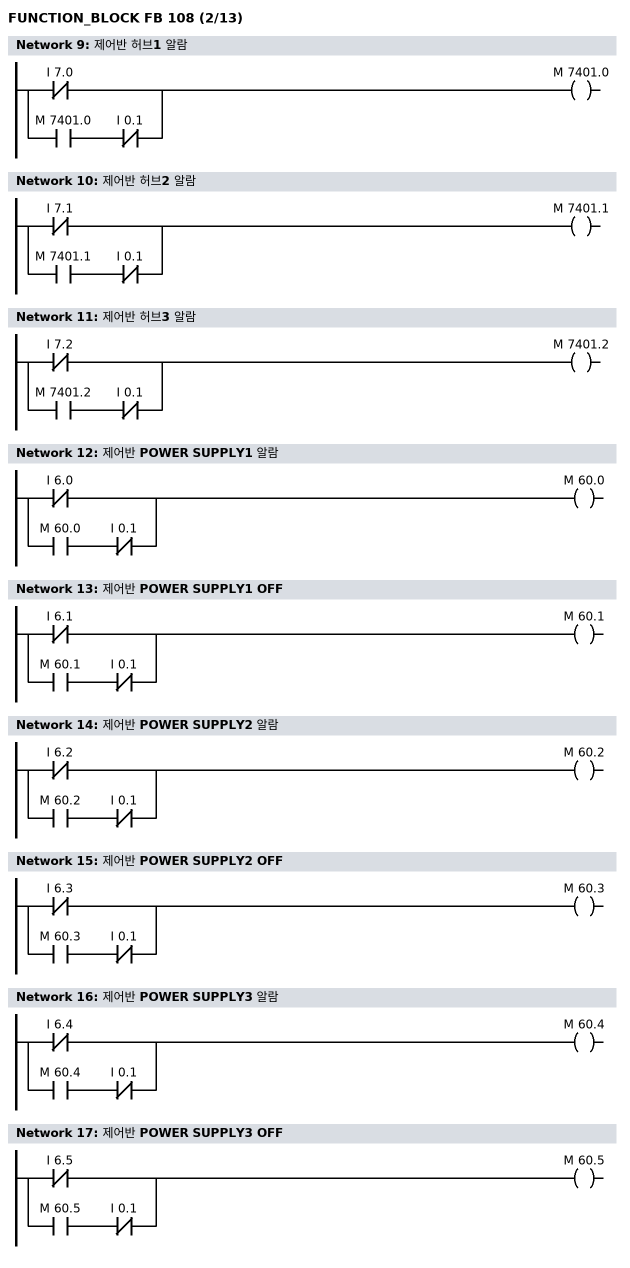

      ON    I      7.0;
      O     ;
      A     M   7401.0;
      AN    I      0.1;
      =     M   7401.0;
NETWORK
TITLE =제어반 허브2 알람

      ON    I      7.1;
      O     ;
      A     M   7401.1;
      AN    I      0.1;
      =     M   7401.1;
NETWORK
TITLE =제어반 허브3 알람

      ON    I      7.2;
      O     ;
      A     M   7401.2;
      AN    I      0.1;
      =     M   7401.2;
NETWORK
TITLE =제어반 POWER SUPPLY1 알람

      ON    I      6.0;
      O     ;
      A     M     60.0;
      AN    I      0.1;
      =     M     60.0;
NETWORK
TITLE =제어반 POWER SUPPLY1 OFF

      ON    I      6.1;
      O     ;
      A     M     60.1;
      AN    I      0.1;
      =     M     60.1;
NETWORK
TITLE =제어반 POWER SUPPLY2 알람
//
//
      ON    I      6.2;
      O     ;
      A     M     60.2;
      AN    I      0.1;
      =     M     60.2;
NETWORK
TITLE =제어반 POWER SUPPLY2 OFF

      ON    I      6.3;
      O     ;
      A     M     60.3;
      AN    I      0.1;
      =     M     60.3;
NETWORK
TITLE =제어반 POWER SUPPLY3 알람
//
//
      ON    I      6.4;
      O     ;
      A     M     60.4;
      AN    I      0.1;
      =     M     60.4;
NETWORK
TITLE =제어반 POWER SUPPLY3 OFF

      ON    I      6.5;
      O     ;
      A     M     60.5;
      AN    I      0.1;
      =     M     60.5;
NETWORK
TITLE =제어반 서지보호기 알람
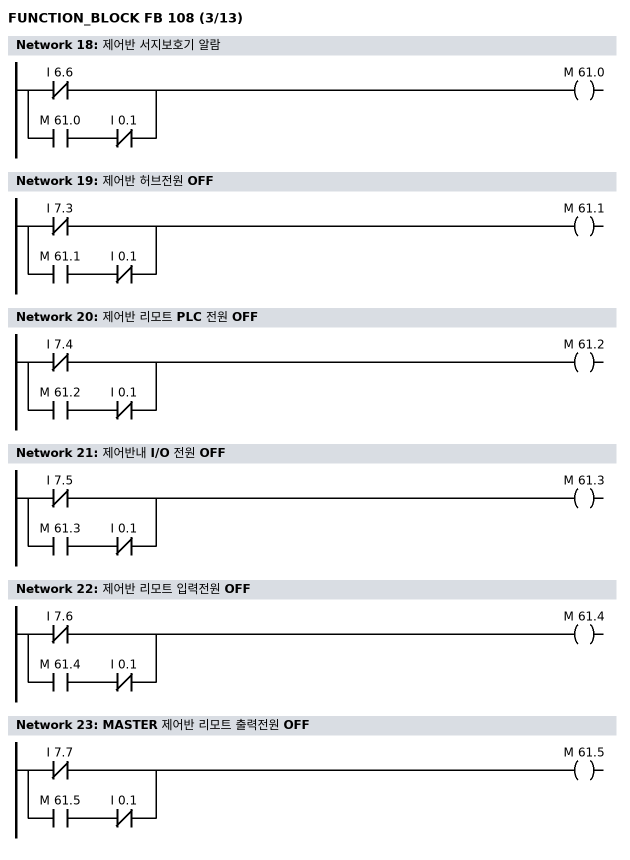

      ON    I      6.6;
      O     ;
      A     M     61.0;
      AN    I      0.1;
      =     M     61.0;
NETWORK
TITLE =제어반 허브전원 OFF

      ON    I      7.3;
      O     ;
      A     M     61.1;
      AN    I      0.1;
      =     M     61.1;
NETWORK
TITLE =제어반 리모트 PLC 전원 OFF

      ON    I      7.4;
      O     ;
      A     M     61.2;
      AN    I      0.1;
      =     M     61.2;
NETWORK
TITLE =제어반내 I/O 전원 OFF

      ON    I      7.5;
      O     ;
      A     M     61.3;
      AN    I      0.1;
      =     M     61.3;
NETWORK
TITLE =제어반 리모트 입력전원 OFF

      ON    I      7.6;
      O     ;
      A     M     61.4;
      AN    I      0.1;
      =     M     61.4;
NETWORK
TITLE =MASTER 제어반 리모트 출력전원 OFF

      ON    I      7.7;
      O     ;
      A     M     61.5;
      AN    I      0.1;
      =     M     61.5;
NETWORK
TITLE =PROFINET ALARM-모듈이상이나 통신케이블단선(1~10)
//
//
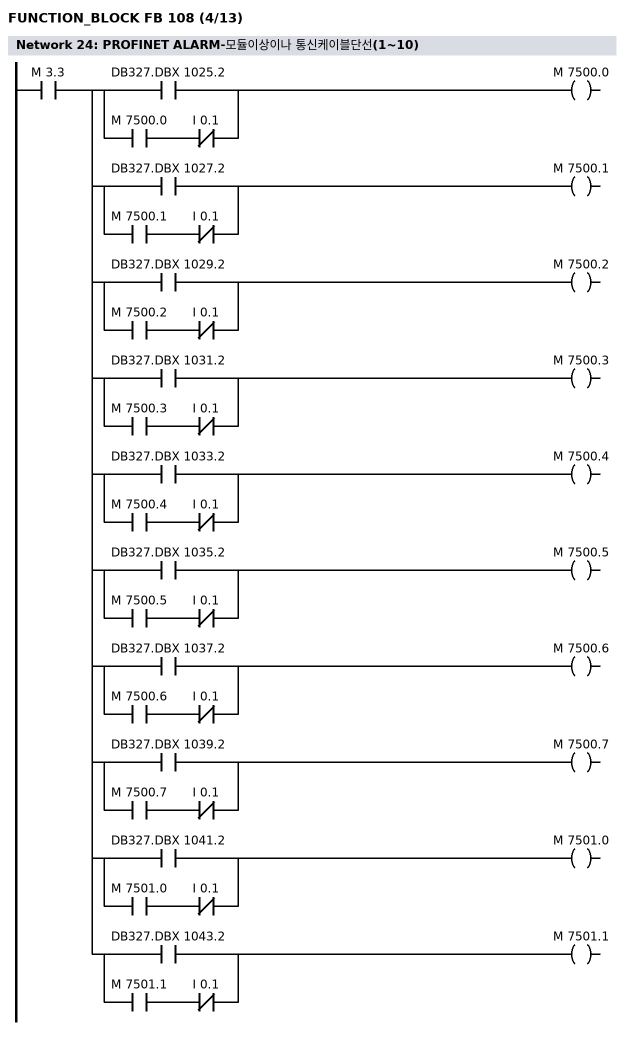
      A     M      3.3;
      =     L      0.0;
      A     L      0.0;
      A(    ;
      O     DB327.DBX 1025.2;
      O     ;
      A     M   7500.0;
      AN    I      0.1;
      )     ;
      =     M   7500.0;
      A     L      0.0;
      A(    ;
      O     DB327.DBX 1027.2;
      O     ;
      A     M   7500.1;
      AN    I      0.1;
      )     ;
      =     M   7500.1;
      A     L      0.0;
      A(    ;
      O     DB327.DBX 1029.2;
      O     ;
      A     M   7500.2;
      AN    I      0.1;
      )     ;
      =     M   7500.2;
      A     L      0.0;
      A(    ;
      O     DB327.DBX 1031.2;
      O     ;
      A     M   7500.3;
      AN    I      0.1;
      )     ;
      =     M   7500.3;
      A     L      0.0;
      A(    ;
      O     DB327.DBX 1033.2;
      O     ;
      A     M   7500.4;
      AN    I      0.1;
      )     ;
      =     M   7500.4;
      A     L      0.0;
      A(    ;
      O     DB327.DBX 1035.2;
      O     ;
      A     M   7500.5;
      AN    I      0.1;
      )     ;
      =     M   7500.5;
      A     L      0.0;
      A(    ;
      O     DB327.DBX 1037.2;
      O     ;
      A     M   7500.6;
      AN    I      0.1;
      )     ;
      =     M   7500.6;
      A     L      0.0;
      A(    ;
      O     DB327.DBX 1039.2;
      O     ;
      A     M   7500.7;
      AN    I      0.1;
      )     ;
      =     M   7500.7;
      A     L      0.0;
      A(    ;
      O     DB327.DBX 1041.2;
      O     ;
      A     M   7501.0;
      AN    I      0.1;
      )     ;
      =     M   7501.0;
      A     L      0.0;
      A(    ;
      O     DB327.DBX 1043.2;
      O     ;
      A     M   7501.1;
      AN    I      0.1;
      )     ;
      =     M   7501.1;
NETWORK
TITLE =PROFINET ALARM-모듈이상이나 통신케이블단선(11~20)
//
//
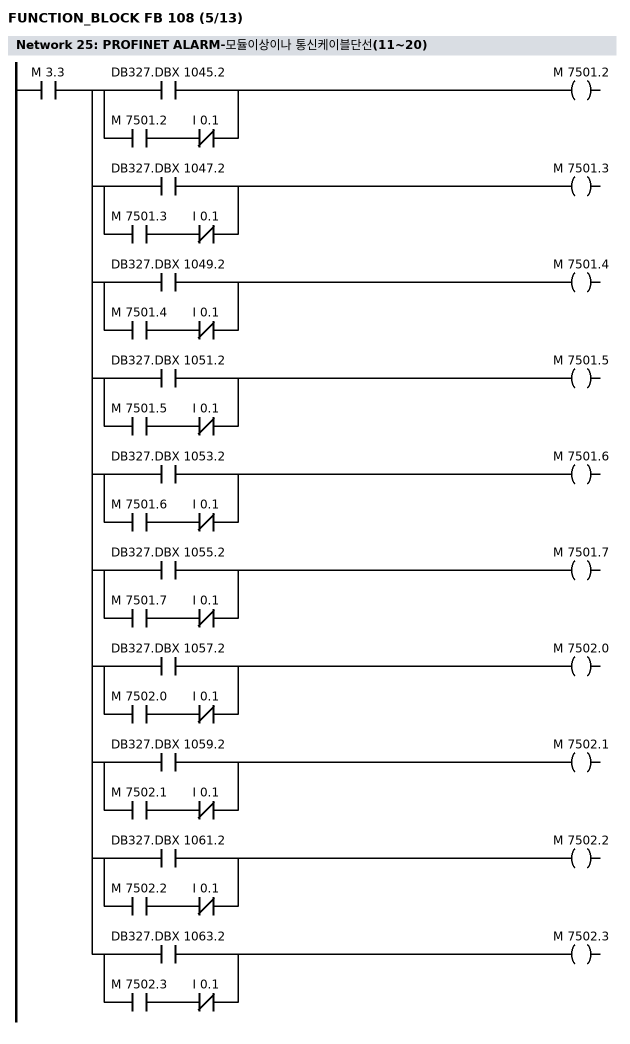
      A     M      3.3;
      =     L      0.0;
      A     L      0.0;
      A(    ;
      O     DB327.DBX 1045.2;
      O     ;
      A     M   7501.2;
      AN    I      0.1;
      )     ;
      =     M   7501.2;
      A     L      0.0;
      A(    ;
      O     DB327.DBX 1047.2;
      O     ;
      A     M   7501.3;
      AN    I      0.1;
      )     ;
      =     M   7501.3;
      A     L      0.0;
      A(    ;
      O     DB327.DBX 1049.2;
      O     ;
      A     M   7501.4;
      AN    I      0.1;
      )     ;
      =     M   7501.4;
      A     L      0.0;
      A(    ;
      O     DB327.DBX 1051.2;
      O     ;
      A     M   7501.5;
      AN    I      0.1;
      )     ;
      =     M   7501.5;
      A     L      0.0;
      A(    ;
      O     DB327.DBX 1053.2;
      O     ;
      A     M   7501.6;
      AN    I      0.1;
      )     ;
      =     M   7501.6;
      A     L      0.0;
      A(    ;
      O     DB327.DBX 1055.2;
      O     ;
      A     M   7501.7;
      AN    I      0.1;
      )     ;
      =     M   7501.7;
      A     L      0.0;
      A(    ;
      O     DB327.DBX 1057.2;
      O     ;
      A     M   7502.0;
      AN    I      0.1;
      )     ;
      =     M   7502.0;
      A     L      0.0;
      A(    ;
      O     DB327.DBX 1059.2;
      O     ;
      A     M   7502.1;
      AN    I      0.1;
      )     ;
      =     M   7502.1;
      A     L      0.0;
      A(    ;
      O     DB327.DBX 1061.2;
      O     ;
      A     M   7502.2;
      AN    I      0.1;
      )     ;
      =     M   7502.2;
      A     L      0.0;
      A(    ;
      O     DB327.DBX 1063.2;
      O     ;
      A     M   7502.3;
      AN    I      0.1;
      )     ;
      =     M   7502.3;
NETWORK
TITLE =PROFINET ALARM-모듈이상이나 통신케이블단선(21~30)
//
//
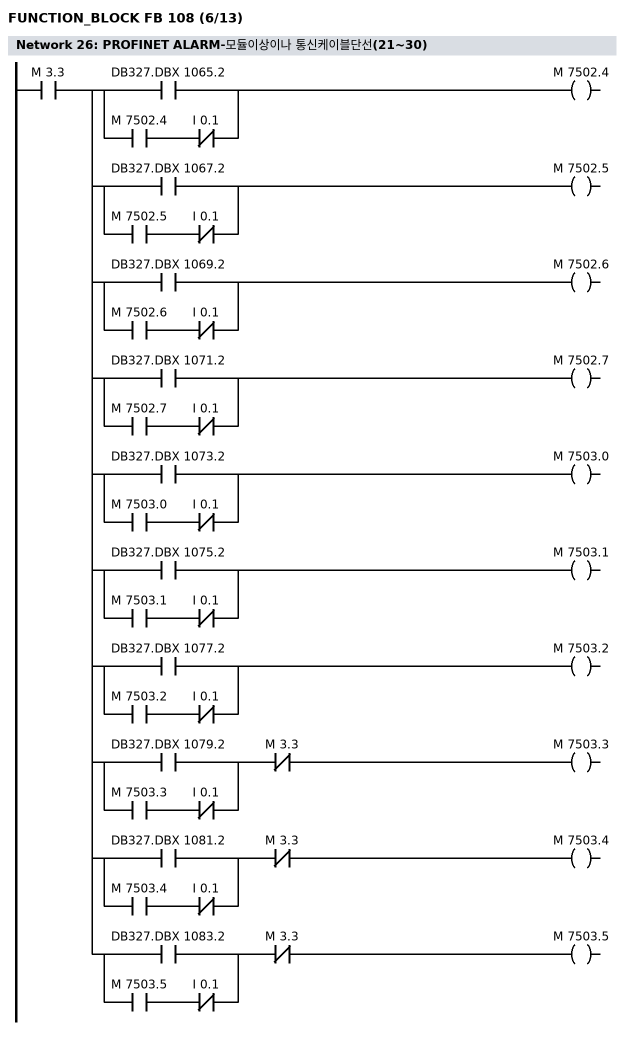
      A     M      3.3;
      =     L      0.0;
      A     L      0.0;
      A(    ;
      O     DB327.DBX 1065.2;
      O     ;
      A     M   7502.4;
      AN    I      0.1;
      )     ;
      =     M   7502.4;
      A     L      0.0;
      A(    ;
      O     DB327.DBX 1067.2;
      O     ;
      A     M   7502.5;
      AN    I      0.1;
      )     ;
      =     M   7502.5;
      A     L      0.0;
      A(    ;
      O     DB327.DBX 1069.2;
      O     ;
      A     M   7502.6;
      AN    I      0.1;
      )     ;
      =     M   7502.6;
      A     L      0.0;
      A(    ;
      O     DB327.DBX 1071.2;
      O     ;
      A     M   7502.7;
      AN    I      0.1;
      )     ;
      =     M   7502.7;
      A     L      0.0;
      A(    ;
      O     DB327.DBX 1073.2;
      O     ;
      A     M   7503.0;
      AN    I      0.1;
      )     ;
      =     M   7503.0;
      A     L      0.0;
      A(    ;
      O     DB327.DBX 1075.2;
      O     ;
      A     M   7503.1;
      AN    I      0.1;
      )     ;
      =     M   7503.1;
      A     L      0.0;
      A(    ;
      O     DB327.DBX 1077.2;
      O     ;
      A     M   7503.2;
      AN    I      0.1;
      )     ;
      =     M   7503.2;
      A     L      0.0;
      A(    ;
      O     DB327.DBX 1079.2;
      O     ;
      A     M   7503.3;
      AN    I      0.1;
      )     ;
      AN    M      3.3;
      =     M   7503.3;
      A     L      0.0;
      A(    ;
      O     DB327.DBX 1081.2;
      O     ;
      A     M   7503.4;
      AN    I      0.1;
      )     ;
      AN    M      3.3;
      =     M   7503.4;
      A     L      0.0;
      A(    ;
      O     DB327.DBX 1083.2;
      O     ;
      A     M   7503.5;
      AN    I      0.1;
      )     ;
      AN    M      3.3;
      =     M   7503.5;
NETWORK
TITLE =PROFINET ALARM-모듈이상이나 통신케이블단선(31~40)
//
//
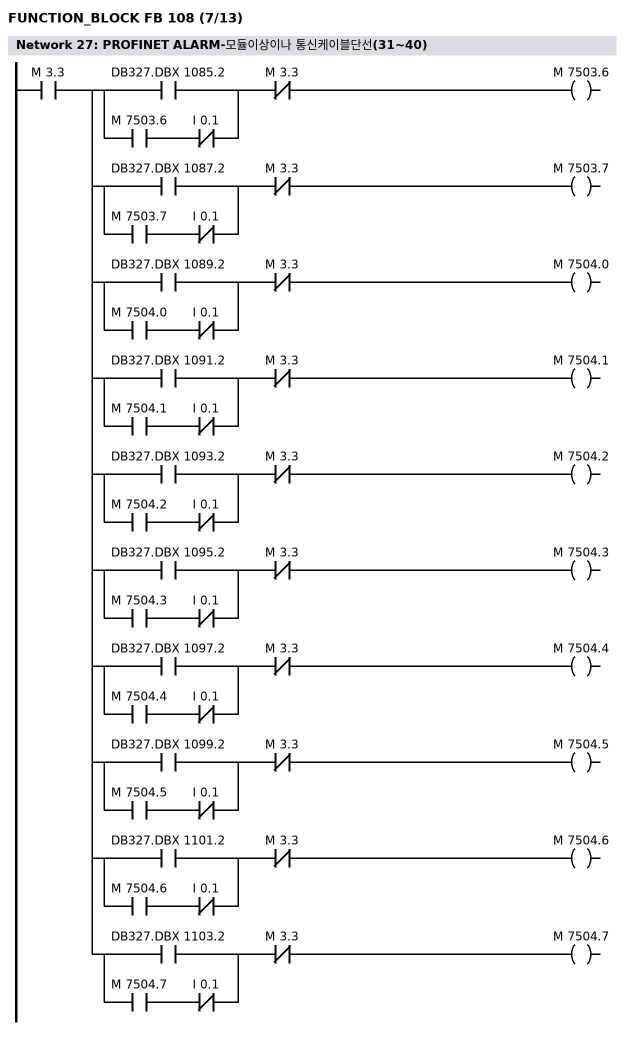
      A     M      3.3;
      =     L      0.0;
      A     L      0.0;
      A(    ;
      O     DB327.DBX 1085.2;
      O     ;
      A     M   7503.6;
      AN    I      0.1;
      )     ;
      AN    M      3.3;
      =     M   7503.6;
      A     L      0.0;
      A(    ;
      O     DB327.DBX 1087.2;
      O     ;
      A     M   7503.7;
      AN    I      0.1;
      )     ;
      AN    M      3.3;
      =     M   7503.7;
      A     L      0.0;
      A(    ;
      O     DB327.DBX 1089.2;
      O     ;
      A     M   7504.0;
      AN    I      0.1;
      )     ;
      AN    M      3.3;
      =     M   7504.0;
      A     L      0.0;
      A(    ;
      O     DB327.DBX 1091.2;
      O     ;
      A     M   7504.1;
      AN    I      0.1;
      )     ;
      AN    M      3.3;
      =     M   7504.1;
      A     L      0.0;
      A(    ;
      O     DB327.DBX 1093.2;
      O     ;
      A     M   7504.2;
      AN    I      0.1;
      )     ;
      AN    M      3.3;
      =     M   7504.2;
      A     L      0.0;
      A(    ;
      O     DB327.DBX 1095.2;
      O     ;
      A     M   7504.3;
      AN    I      0.1;
      )     ;
      AN    M      3.3;
      =     M   7504.3;
      A     L      0.0;
      A(    ;
      O     DB327.DBX 1097.2;
      O     ;
      A     M   7504.4;
      AN    I      0.1;
      )     ;
      AN    M      3.3;
      =     M   7504.4;
      A     L      0.0;
      A(    ;
      O     DB327.DBX 1099.2;
      O     ;
      A     M   7504.5;
      AN    I      0.1;
      )     ;
      AN    M      3.3;
      =     M   7504.5;
      A     L      0.0;
      A(    ;
      O     DB327.DBX 1101.2;
      O     ;
      A     M   7504.6;
      AN    I      0.1;
      )     ;
      AN    M      3.3;
      =     M   7504.6;
      A     L      0.0;
      A(    ;
      O     DB327.DBX 1103.2;
      O     ;
      A     M   7504.7;
      AN    I      0.1;
      )     ;
      AN    M      3.3;
      =     M   7504.7;
NETWORK
TITLE =PROFINET ALARM-모듈이상이나 통신케이블단선(150~159)
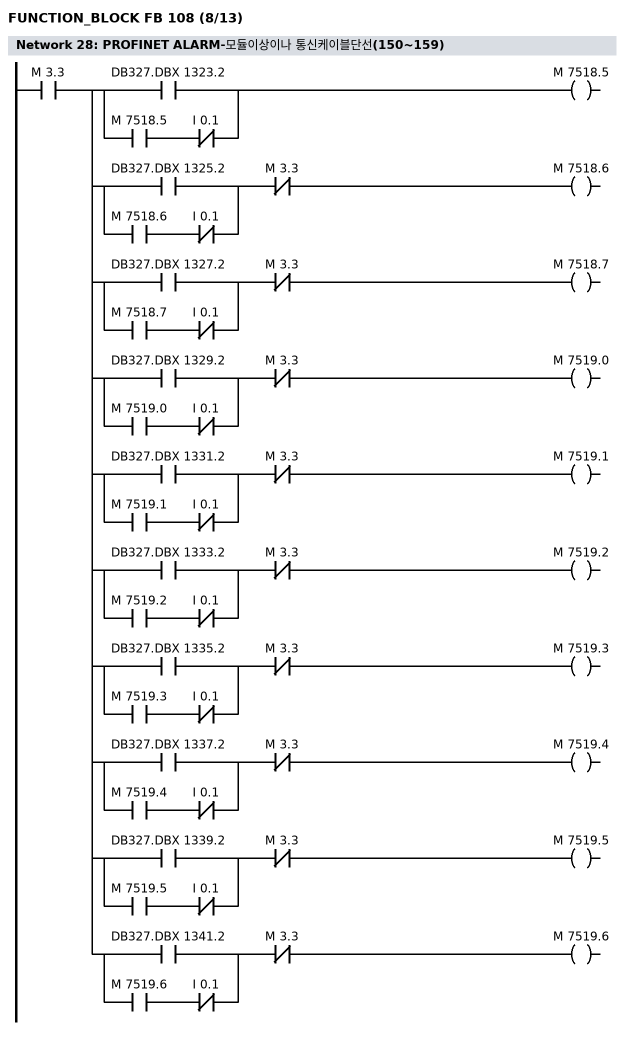

      A     M      3.3;
      =     L      0.0;
      A     L      0.0;
      A(    ;
      O     DB327.DBX 1323.2;
      O     ;
      A     M   7518.5;
      AN    I      0.1;
      )     ;
      =     M   7518.5;
      A     L      0.0;
      A(    ;
      O     DB327.DBX 1325.2;
      O     ;
      A     M   7518.6;
      AN    I      0.1;
      )     ;
      AN    M      3.3;
      =     M   7518.6;
      A     L      0.0;
      A(    ;
      O     DB327.DBX 1327.2;
      O     ;
      A     M   7518.7;
      AN    I      0.1;
      )     ;
      AN    M      3.3;
      =     M   7518.7;
      A     L      0.0;
      A(    ;
      O     DB327.DBX 1329.2;
      O     ;
      A     M   7519.0;
      AN    I      0.1;
      )     ;
      AN    M      3.3;
      =     M   7519.0;
      A     L      0.0;
      A(    ;
      O     DB327.DBX 1331.2;
      O     ;
      A     M   7519.1;
      AN    I      0.1;
      )     ;
      AN    M      3.3;
      =     M   7519.1;
      A     L      0.0;
      A(    ;
      O     DB327.DBX 1333.2;
      O     ;
      A     M   7519.2;
      AN    I      0.1;
      )     ;
      AN    M      3.3;
      =     M   7519.2;
      A     L      0.0;
      A(    ;
      O     DB327.DBX 1335.2;
      O     ;
      A     M   7519.3;
      AN    I      0.1;
      )     ;
      AN    M      3.3;
      =     M   7519.3;
      A     L      0.0;
      A(    ;
      O     DB327.DBX 1337.2;
      O     ;
      A     M   7519.4;
      AN    I      0.1;
      )     ;
      AN    M      3.3;
      =     M   7519.4;
      A     L      0.0;
      A(    ;
      O     DB327.DBX 1339.2;
      O     ;
      A     M   7519.5;
      AN    I      0.1;
      )     ;
      AN    M      3.3;
      =     M   7519.5;
      A     L      0.0;
      A(    ;
      O     DB327.DBX 1341.2;
      O     ;
      A     M   7519.6;
      AN    I      0.1;
      )     ;
      AN    M      3.3;
      =     M   7519.6;
NETWORK
TITLE =PROFINET MODULE ERROR(1~10)
//
//
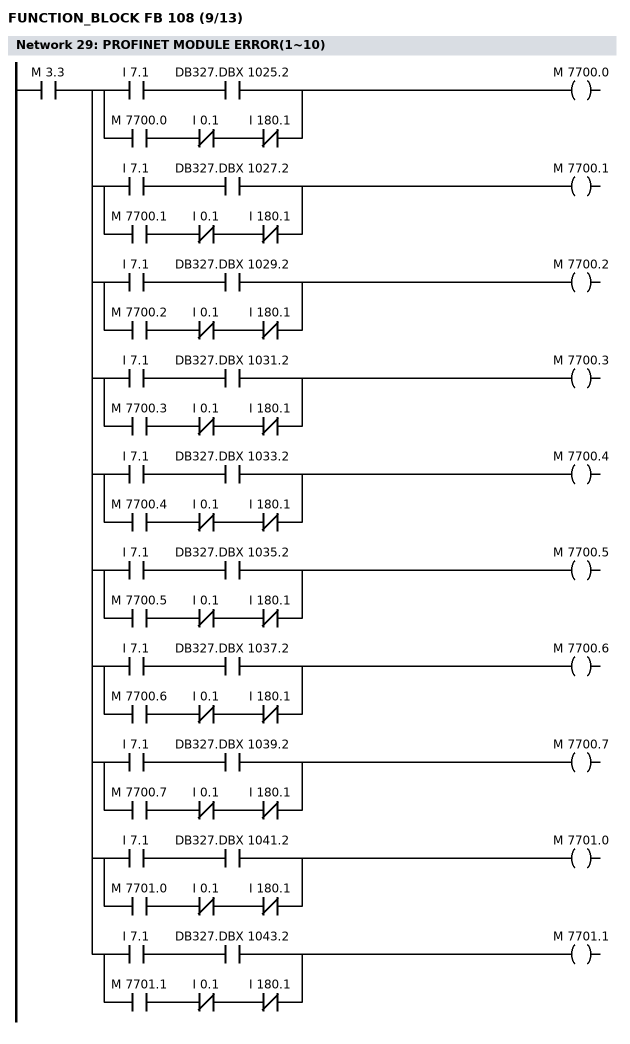
      A     M      3.3;
      =     L      0.0;
      A     L      0.0;
      A(    ;
      A     I      7.1;
      A     DB327.DBX 1025.2;
      O     ;
      A     M   7700.0;
      AN    I      0.1;
      AN    I    180.1;
      )     ;
      =     M   7700.0;
      A     L      0.0;
      A(    ;
      A     I      7.1;
      A     DB327.DBX 1027.2;
      O     ;
      A     M   7700.1;
      AN    I      0.1;
      AN    I    180.1;
      )     ;
      =     M   7700.1;
      A     L      0.0;
      A(    ;
      A     I      7.1;
      A     DB327.DBX 1029.2;
      O     ;
      A     M   7700.2;
      AN    I      0.1;
      AN    I    180.1;
      )     ;
      =     M   7700.2;
      A     L      0.0;
      A(    ;
      A     I      7.1;
      A     DB327.DBX 1031.2;
      O     ;
      A     M   7700.3;
      AN    I      0.1;
      AN    I    180.1;
      )     ;
      =     M   7700.3;
      A     L      0.0;
      A(    ;
      A     I      7.1;
      A     DB327.DBX 1033.2;
      O     ;
      A     M   7700.4;
      AN    I      0.1;
      AN    I    180.1;
      )     ;
      =     M   7700.4;
      A     L      0.0;
      A(    ;
      A     I      7.1;
      A     DB327.DBX 1035.2;
      O     ;
      A     M   7700.5;
      AN    I      0.1;
      AN    I    180.1;
      )     ;
      =     M   7700.5;
      A     L      0.0;
      A(    ;
      A     I      7.1;
      A     DB327.DBX 1037.2;
      O     ;
      A     M   7700.6;
      AN    I      0.1;
      AN    I    180.1;
      )     ;
      =     M   7700.6;
      A     L      0.0;
      A(    ;
      A     I      7.1;
      A     DB327.DBX 1039.2;
      O     ;
      A     M   7700.7;
      AN    I      0.1;
      AN    I    180.1;
      )     ;
      =     M   7700.7;
      A     L      0.0;
      A(    ;
      A     I      7.1;
      A     DB327.DBX 1041.2;
      O     ;
      A     M   7701.0;
      AN    I      0.1;
      AN    I    180.1;
      )     ;
      =     M   7701.0;
      A     L      0.0;
      A(    ;
      A     I      7.1;
      A     DB327.DBX 1043.2;
      O     ;
      A     M   7701.1;
      AN    I      0.1;
      AN    I    180.1;
      )     ;
      =     M   7701.1;
NETWORK
TITLE =PROFINET MODULE ERROR(11~20)
//
//
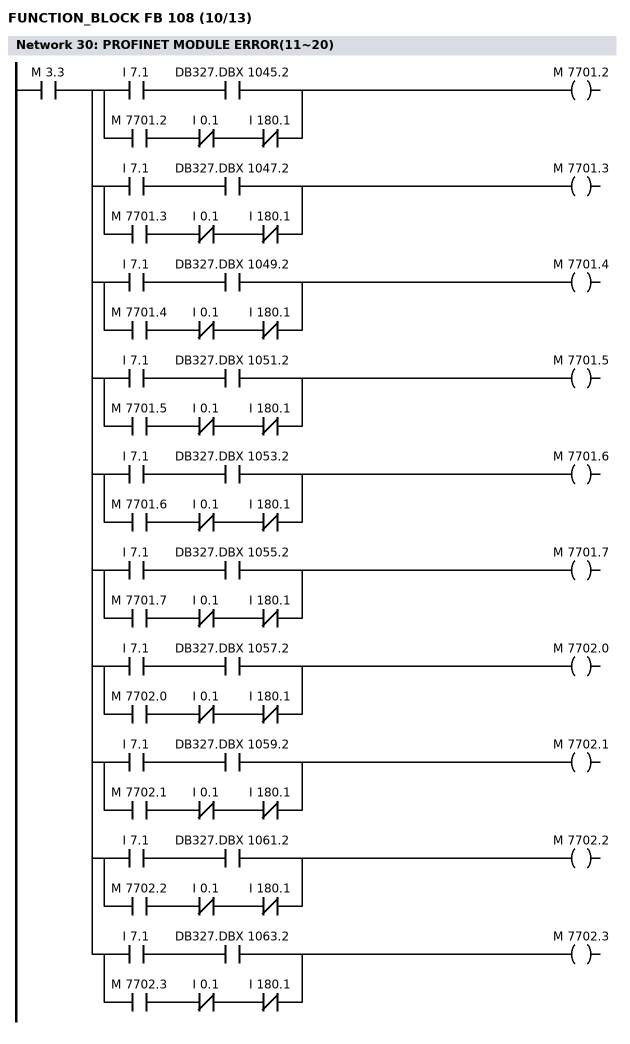
      A     M      3.3;
      =     L      0.0;
      A     L      0.0;
      A(    ;
      A     I      7.1;
      A     DB327.DBX 1045.2;
      O     ;
      A     M   7701.2;
      AN    I      0.1;
      AN    I    180.1;
      )     ;
      =     M   7701.2;
      A     L      0.0;
      A(    ;
      A     I      7.1;
      A     DB327.DBX 1047.2;
      O     ;
      A     M   7701.3;
      AN    I      0.1;
      AN    I    180.1;
      )     ;
      =     M   7701.3;
      A     L      0.0;
      A(    ;
      A     I      7.1;
      A     DB327.DBX 1049.2;
      O     ;
      A     M   7701.4;
      AN    I      0.1;
      AN    I    180.1;
      )     ;
      =     M   7701.4;
      A     L      0.0;
      A(    ;
      A     I      7.1;
      A     DB327.DBX 1051.2;
      O     ;
      A     M   7701.5;
      AN    I      0.1;
      AN    I    180.1;
      )     ;
      =     M   7701.5;
      A     L      0.0;
      A(    ;
      A     I      7.1;
      A     DB327.DBX 1053.2;
      O     ;
      A     M   7701.6;
      AN    I      0.1;
      AN    I    180.1;
      )     ;
      =     M   7701.6;
      A     L      0.0;
      A(    ;
      A     I      7.1;
      A     DB327.DBX 1055.2;
      O     ;
      A     M   7701.7;
      AN    I      0.1;
      AN    I    180.1;
      )     ;
      =     M   7701.7;
      A     L      0.0;
      A(    ;
      A     I      7.1;
      A     DB327.DBX 1057.2;
      O     ;
      A     M   7702.0;
      AN    I      0.1;
      AN    I    180.1;
      )     ;
      =     M   7702.0;
      A     L      0.0;
      A(    ;
      A     I      7.1;
      A     DB327.DBX 1059.2;
      O     ;
      A     M   7702.1;
      AN    I      0.1;
      AN    I    180.1;
      )     ;
      =     M   7702.1;
      A     L      0.0;
      A(    ;
      A     I      7.1;
      A     DB327.DBX 1061.2;
      O     ;
      A     M   7702.2;
      AN    I      0.1;
      AN    I    180.1;
      )     ;
      =     M   7702.2;
      A     L      0.0;
      A(    ;
      A     I      7.1;
      A     DB327.DBX 1063.2;
      O     ;
      A     M   7702.3;
      AN    I      0.1;
      AN    I    180.1;
      )     ;
      =     M   7702.3;
NETWORK
TITLE =PROFINET MODULE ERROR(21~30)
//
//
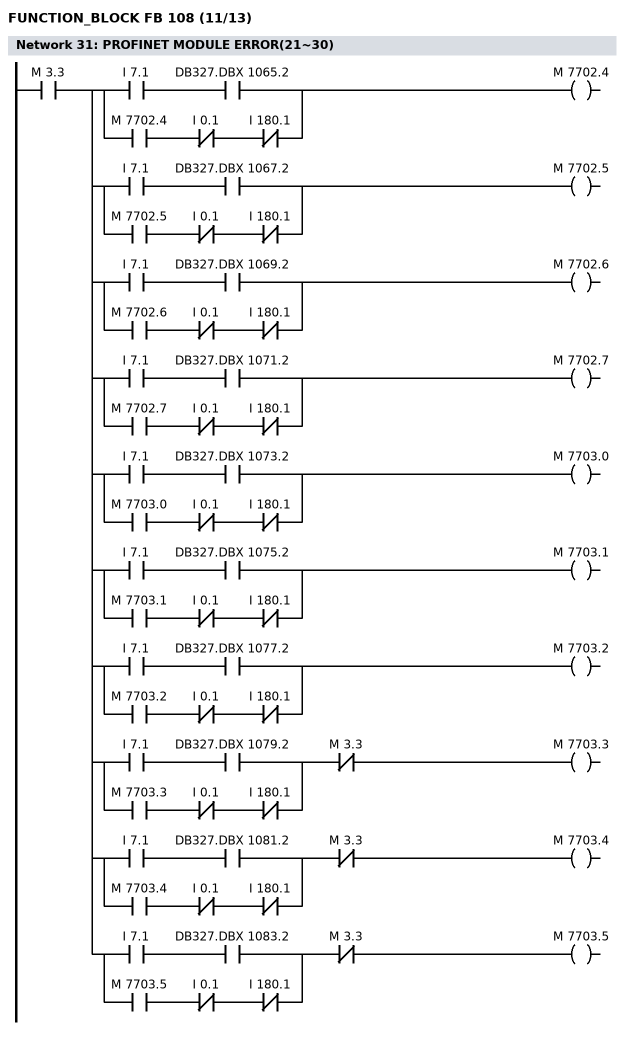
      A     M      3.3;
      =     L      0.0;
      A     L      0.0;
      A(    ;
      A     I      7.1;
      A     DB327.DBX 1065.2;
      O     ;
      A     M   7702.4;
      AN    I      0.1;
      AN    I    180.1;
      )     ;
      =     M   7702.4;
      A     L      0.0;
      A(    ;
      A     I      7.1;
      A     DB327.DBX 1067.2;
      O     ;
      A     M   7702.5;
      AN    I      0.1;
      AN    I    180.1;
      )     ;
      =     M   7702.5;
      A     L      0.0;
      A(    ;
      A     I      7.1;
      A     DB327.DBX 1069.2;
      O     ;
      A     M   7702.6;
      AN    I      0.1;
      AN    I    180.1;
      )     ;
      =     M   7702.6;
      A     L      0.0;
      A(    ;
      A     I      7.1;
      A     DB327.DBX 1071.2;
      O     ;
      A     M   7702.7;
      AN    I      0.1;
      AN    I    180.1;
      )     ;
      =     M   7702.7;
      A     L      0.0;
      A(    ;
      A     I      7.1;
      A     DB327.DBX 1073.2;
      O     ;
      A     M   7703.0;
      AN    I      0.1;
      AN    I    180.1;
      )     ;
      =     M   7703.0;
      A     L      0.0;
      A(    ;
      A     I      7.1;
      A     DB327.DBX 1075.2;
      O     ;
      A     M   7703.1;
      AN    I      0.1;
      AN    I    180.1;
      )     ;
      =     M   7703.1;
      A     L      0.0;
      A(    ;
      A     I      7.1;
      A     DB327.DBX 1077.2;
      O     ;
      A     M   7703.2;
      AN    I      0.1;
      AN    I    180.1;
      )     ;
      =     M   7703.2;
      A     L      0.0;
      A(    ;
      A     I      7.1;
      A     DB327.DBX 1079.2;
      O     ;
      A     M   7703.3;
      AN    I      0.1;
      AN    I    180.1;
      )     ;
      AN    M      3.3;
      =     M   7703.3;
      A     L      0.0;
      A(    ;
      A     I      7.1;
      A     DB327.DBX 1081.2;
      O     ;
      A     M   7703.4;
      AN    I      0.1;
      AN    I    180.1;
      )     ;
      AN    M      3.3;
      =     M   7703.4;
      A     L      0.0;
      A(    ;
      A     I      7.1;
      A     DB327.DBX 1083.2;
      O     ;
      A     M   7703.5;
      AN    I      0.1;
      AN    I    180.1;
      )     ;
      AN    M      3.3;
      =     M   7703.5;
NETWORK
TITLE =PROFINET MODULE ERROR(31~40)
//
//
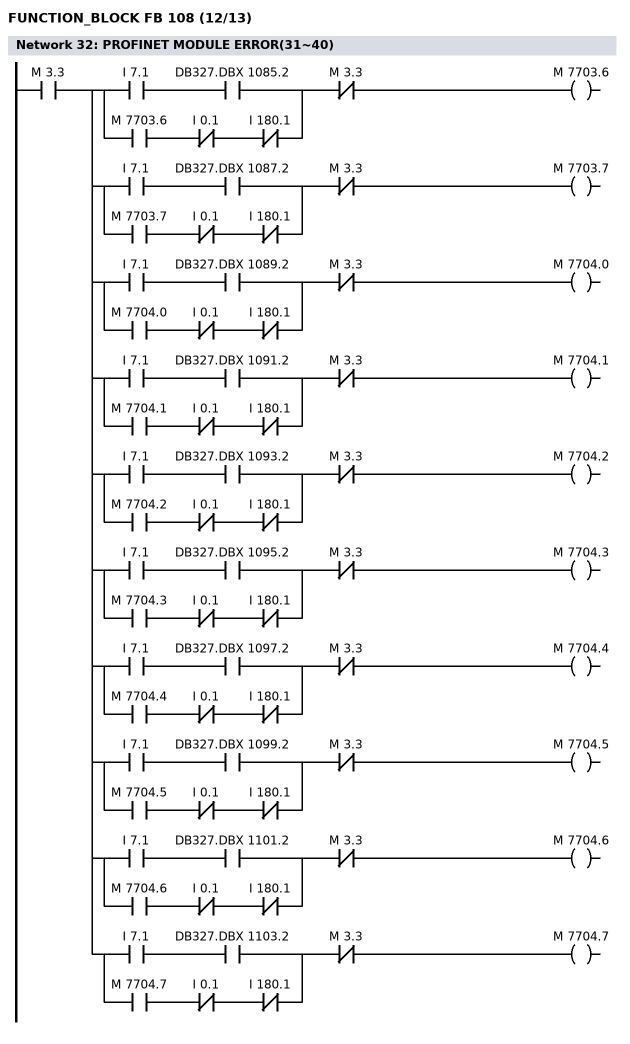
      A     M      3.3;
      =     L      0.0;
      A     L      0.0;
      A(    ;
      A     I      7.1;
      A     DB327.DBX 1085.2;
      O     ;
      A     M   7703.6;
      AN    I      0.1;
      AN    I    180.1;
      )     ;
      AN    M      3.3;
      =     M   7703.6;
      A     L      0.0;
      A(    ;
      A     I      7.1;
      A     DB327.DBX 1087.2;
      O     ;
      A     M   7703.7;
      AN    I      0.1;
      AN    I    180.1;
      )     ;
      AN    M      3.3;
      =     M   7703.7;
      A     L      0.0;
      A(    ;
      A     I      7.1;
      A     DB327.DBX 1089.2;
      O     ;
      A     M   7704.0;
      AN    I      0.1;
      AN    I    180.1;
      )     ;
      AN    M      3.3;
      =     M   7704.0;
      A     L      0.0;
      A(    ;
      A     I      7.1;
      A     DB327.DBX 1091.2;
      O     ;
      A     M   7704.1;
      AN    I      0.1;
      AN    I    180.1;
      )     ;
      AN    M      3.3;
      =     M   7704.1;
      A     L      0.0;
      A(    ;
      A     I      7.1;
      A     DB327.DBX 1093.2;
      O     ;
      A     M   7704.2;
      AN    I      0.1;
      AN    I    180.1;
      )     ;
      AN    M      3.3;
      =     M   7704.2;
      A     L      0.0;
      A(    ;
      A     I      7.1;
      A     DB327.DBX 1095.2;
      O     ;
      A     M   7704.3;
      AN    I      0.1;
      AN    I    180.1;
      )     ;
      AN    M      3.3;
      =     M   7704.3;
      A     L      0.0;
      A(    ;
      A     I      7.1;
      A     DB327.DBX 1097.2;
      O     ;
      A     M   7704.4;
      AN    I      0.1;
      AN    I    180.1;
      )     ;
      AN    M      3.3;
      =     M   7704.4;
      A     L      0.0;
      A(    ;
      A     I      7.1;
      A     DB327.DBX 1099.2;
      O     ;
      A     M   7704.5;
      AN    I      0.1;
      AN    I    180.1;
      )     ;
      AN    M      3.3;
      =     M   7704.5;
      A     L      0.0;
      A(    ;
      A     I      7.1;
      A     DB327.DBX 1101.2;
      O     ;
      A     M   7704.6;
      AN    I      0.1;
      AN    I    180.1;
      )     ;
      AN    M      3.3;
      =     M   7704.6;
      A     L      0.0;
      A(    ;
      A     I      7.1;
      A     DB327.DBX 1103.2;
      O     ;
      A     M   7704.7;
      AN    I      0.1;
      AN    I    180.1;
      )     ;
      AN    M      3.3;
      =     M   7704.7;
NETWORK
TITLE =PROFINET MODULE ERROR(150~159)
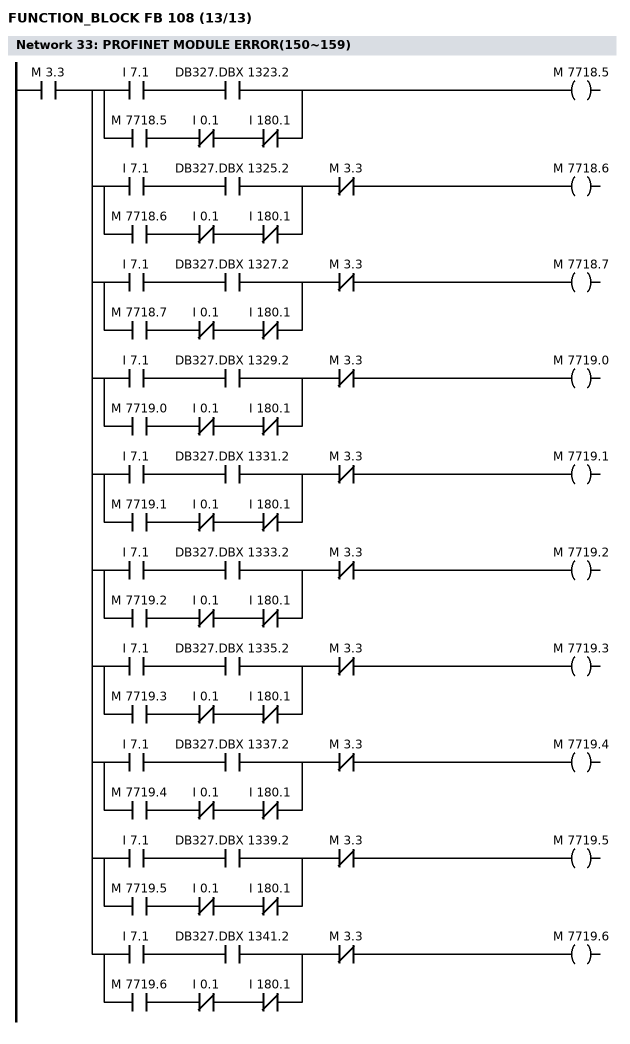

      A     M      3.3;
      =     L      0.0;
      A     L      0.0;
      A(    ;
      A     I      7.1;
      A     DB327.DBX 1323.2;
      O     ;
      A     M   7718.5;
      AN    I      0.1;
      AN    I    180.1;
      )     ;
      =     M   7718.5;
      A     L      0.0;
      A(    ;
      A     I      7.1;
      A     DB327.DBX 1325.2;
      O     ;
      A     M   7718.6;
      AN    I      0.1;
      AN    I    180.1;
      )     ;
      AN    M      3.3;
      =     M   7718.6;
      A     L      0.0;
      A(    ;
      A     I      7.1;
      A     DB327.DBX 1327.2;
      O     ;
      A     M   7718.7;
      AN    I      0.1;
      AN    I    180.1;
      )     ;
      AN    M      3.3;
      =     M   7718.7;
      A     L      0.0;
      A(    ;
      A     I      7.1;
      A     DB327.DBX 1329.2;
      O     ;
      A     M   7719.0;
      AN    I      0.1;
      AN    I    180.1;
      )     ;
      AN    M      3.3;
      =     M   7719.0;
      A     L      0.0;
      A(    ;
      A     I      7.1;
      A     DB327.DBX 1331.2;
      O     ;
      A     M   7719.1;
      AN    I      0.1;
      AN    I    180.1;
      )     ;
      AN    M      3.3;
      =     M   7719.1;
      A     L      0.0;
      A(    ;
      A     I      7.1;
      A     DB327.DBX 1333.2;
      O     ;
      A     M   7719.2;
      AN    I      0.1;
      AN    I    180.1;
      )     ;
      AN    M      3.3;
      =     M   7719.2;
      A     L      0.0;
      A(    ;
      A     I      7.1;
      A     DB327.DBX 1335.2;
      O     ;
      A     M   7719.3;
      AN    I      0.1;
      AN    I    180.1;
      )     ;
      AN    M      3.3;
      =     M   7719.3;
      A     L      0.0;
      A(    ;
      A     I      7.1;
      A     DB327.DBX 1337.2;
      O     ;
      A     M   7719.4;
      AN    I      0.1;
      AN    I    180.1;
      )     ;
      AN    M      3.3;
      =     M   7719.4;
      A     L      0.0;
      A(    ;
      A     I      7.1;
      A     DB327.DBX 1339.2;
      O     ;
      A     M   7719.5;
      AN    I      0.1;
      AN    I    180.1;
      )     ;
      AN    M      3.3;
      =     M   7719.5;
      A     L      0.0;
      A(    ;
      A     I      7.1;
      A     DB327.DBX 1341.2;
      O     ;
      A     M   7719.6;
      AN    I      0.1;
      AN    I    180.1;
      )     ;
      AN    M      3.3;
      =     M   7719.6;
END_FUNCTION_BLOCK

DATA_BLOCK DB 108
TITLE =
VERSION : 0.0

 FB 108
BEGIN
END_DATA_BLOCK

FUNCTION_BLOCK FB 110
TITLE =
VERSION : 0.1


VAR
  S700_1_STN_MODE : FB 402;	//S700_1_STN_MODE
END_VAR
BEGIN
NETWORK
TITLE =
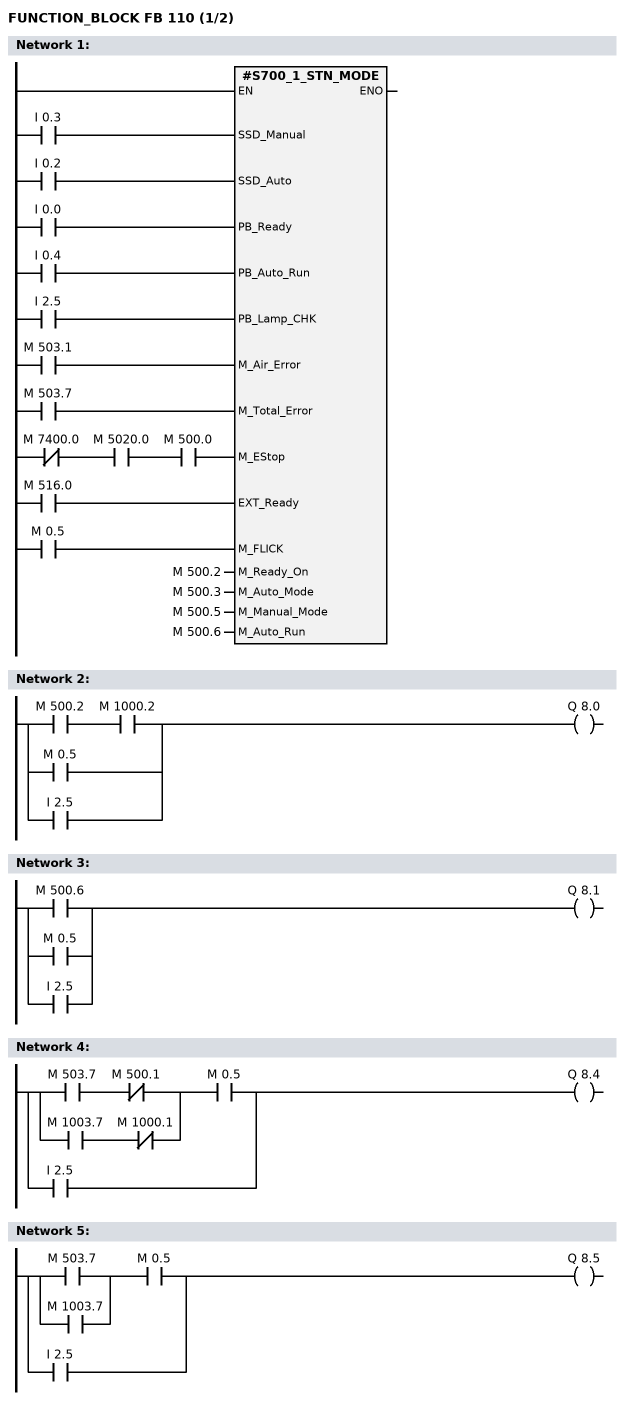

      A     I      0.3;
      =     L      0.0;
      BLD   103;
      A     I      0.2;
      =     L      0.1;
      BLD   103;
      A     I      0.0;
      =     L      0.2;
      BLD   103;
      A     I      0.4;
      =     L      0.3;
      BLD   103;
      A     I      2.5;
      =     L      0.6;
      BLD   103;
      A     M    503.1;
      =     L      0.7;
      BLD   103;
      A     M    503.7;
      =     L      1.1;
      BLD   103;
      AN    M   7400.0;
      A     M   5020.0;
      A     M    500.0;
      =     L      1.2;
      BLD   103;
      A     M    516.0;
      =     L      1.3;
      BLD   103;
      A     M      0.5;
      =     L      1.5;
      BLD   103;
      CALL #S700_1_STN_MODE (
           SSD_Manual               := L      0.0,
           SSD_Auto                 := L      0.1,
           PB_Ready                 := L      0.2,
           PB_Auto_Run              := L      0.3,
           PB_Lamp_CHK              := L      0.6,
           M_Air_Error              := L      0.7,
           M_Total_Error            := L      1.1,
           M_EStop                  := L      1.2,
           EXT_Ready                := L      1.3,
           M_FLICK                  := L      1.5,
           M_Ready_On               := M    500.2,
           M_Auto_Mode              := M    500.3,
           M_Manual_Mode            := M    500.5,
           M_Auto_Run               := M    500.6);

      NOP   0;
NETWORK
TITLE =

      A     M    500.2;
      A     M   1000.2;
      O     M      0.5;
      O     I      2.5;
      =     Q      8.0;
NETWORK
TITLE =

      O     M    500.6;
      O     M      0.5;
      O     I      2.5;
      =     Q      8.1;
NETWORK
TITLE =

      A(    ;
      A     M    503.7;
      AN    M    500.1;
      O     ;
      A     M   1003.7;
      AN    M   1000.1;
      )     ;
      A     M      0.5;
      O     I      2.5;
      =     Q      8.4;
NETWORK
TITLE =

      A(    ;
      O     M    503.7;
      O     M   1003.7;
      )     ;
      A     M      0.5;
      O     I      2.5;
      =     Q      8.5;
NETWORK
TITLE =
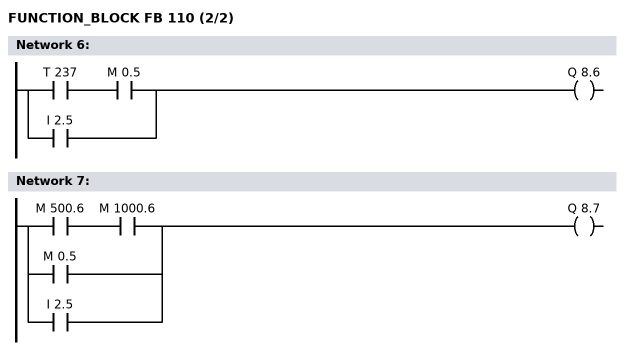

      A     T    237;
      A     M      0.5;
      O     I      2.5;
      =     Q      8.6;
NETWORK
TITLE =

      A     M    500.6;
      A     M   1000.6;
      O     M      0.5;
      O     I      2.5;
      =     Q      8.7;
END_FUNCTION_BLOCK

DATA_BLOCK DB 110
TITLE =
VERSION : 0.0

 FB 110
BEGIN
   S700_1_STN_MODE.SSD_Manual := FALSE;
   S700_1_STN_MODE.SSD_Auto := FALSE;
   S700_1_STN_MODE.PB_Ready := FALSE;
   S700_1_STN_MODE.PB_Auto_Run := FALSE;
   S700_1_STN_MODE.PB_Remote_Ready := FALSE;
   S700_1_STN_MODE.PB_Remote_Auto_Run := FALSE;
   S700_1_STN_MODE.PB_Lamp_CHK := FALSE;
   S700_1_STN_MODE.M_Air_Error := FALSE;
   S700_1_STN_MODE.M_Water_Error := FALSE;
   S700_1_STN_MODE.M_Total_Error := FALSE;
   S700_1_STN_MODE.M_EStop := FALSE;
   S700_1_STN_MODE.EXT_Ready := FALSE;
   S700_1_STN_MODE.EXT_Auto := FALSE;
   S700_1_STN_MODE.T_SemiAuto := T#0MS;
   S700_1_STN_MODE.M_FLICK := FALSE;
   S700_1_STN_MODE.M_Ready_On := FALSE;
   S700_1_STN_MODE.M_Auto_Mode := FALSE;
   S700_1_STN_MODE.M_SemiAuto_Mode := FALSE;
   S700_1_STN_MODE.M_Manual_Mode := FALSE;
   S700_1_STN_MODE.M_Auto_Run := FALSE;
   S700_1_STN_MODE.LP_Ready_On := FALSE;
   S700_1_STN_MODE.LP_Auto_Run := FALSE;
   S700_1_STN_MODE.AUTO_MODE_DELAY.IN := FALSE;
   S700_1_STN_MODE.AUTO_MODE_DELAY.PT := T#0MS;
   S700_1_STN_MODE.AUTO_MODE_DELAY.Q := FALSE;
   S700_1_STN_MODE.AUTO_MODE_DELAY.ET := T#0MS;
   S700_1_STN_MODE.AUTO_MODE_DELAY.STATE := B#16#0;
   S700_1_STN_MODE.AUTO_MODE_DELAY.STIME := T#0MS;
   S700_1_STN_MODE.AUTO_MODE_DELAY.ATIME := T#0MS;
   S700_1_STN_MODE.SEMI_AUTO_DELAY.IN := FALSE;
   S700_1_STN_MODE.SEMI_AUTO_DELAY.PT := T#0MS;
   S700_1_STN_MODE.SEMI_AUTO_DELAY.Q := FALSE;
   S700_1_STN_MODE.SEMI_AUTO_DELAY.ET := T#0MS;
   S700_1_STN_MODE.SEMI_AUTO_DELAY.STATE := B#16#0;
   S700_1_STN_MODE.SEMI_AUTO_DELAY.STIME := T#0MS;
   S700_1_STN_MODE.SEMI_AUTO_DELAY.ATIME := T#0MS;
   S700_1_STN_MODE.MANUAL_DELAY.IN := FALSE;
   S700_1_STN_MODE.MANUAL_DELAY.PT := T#0MS;
   S700_1_STN_MODE.MANUAL_DELAY.Q := FALSE;
   S700_1_STN_MODE.MANUAL_DELAY.ET := T#0MS;
   S700_1_STN_MODE.MANUAL_DELAY.STATE := B#16#0;
   S700_1_STN_MODE.MANUAL_DELAY.STIME := T#0MS;
   S700_1_STN_MODE.MANUAL_DELAY.ATIME := T#0MS;
END_DATA_BLOCK

FUNCTION FC 110 : VOID
TITLE =
VERSION : 0.1

BEGIN
NETWORK
TITLE =
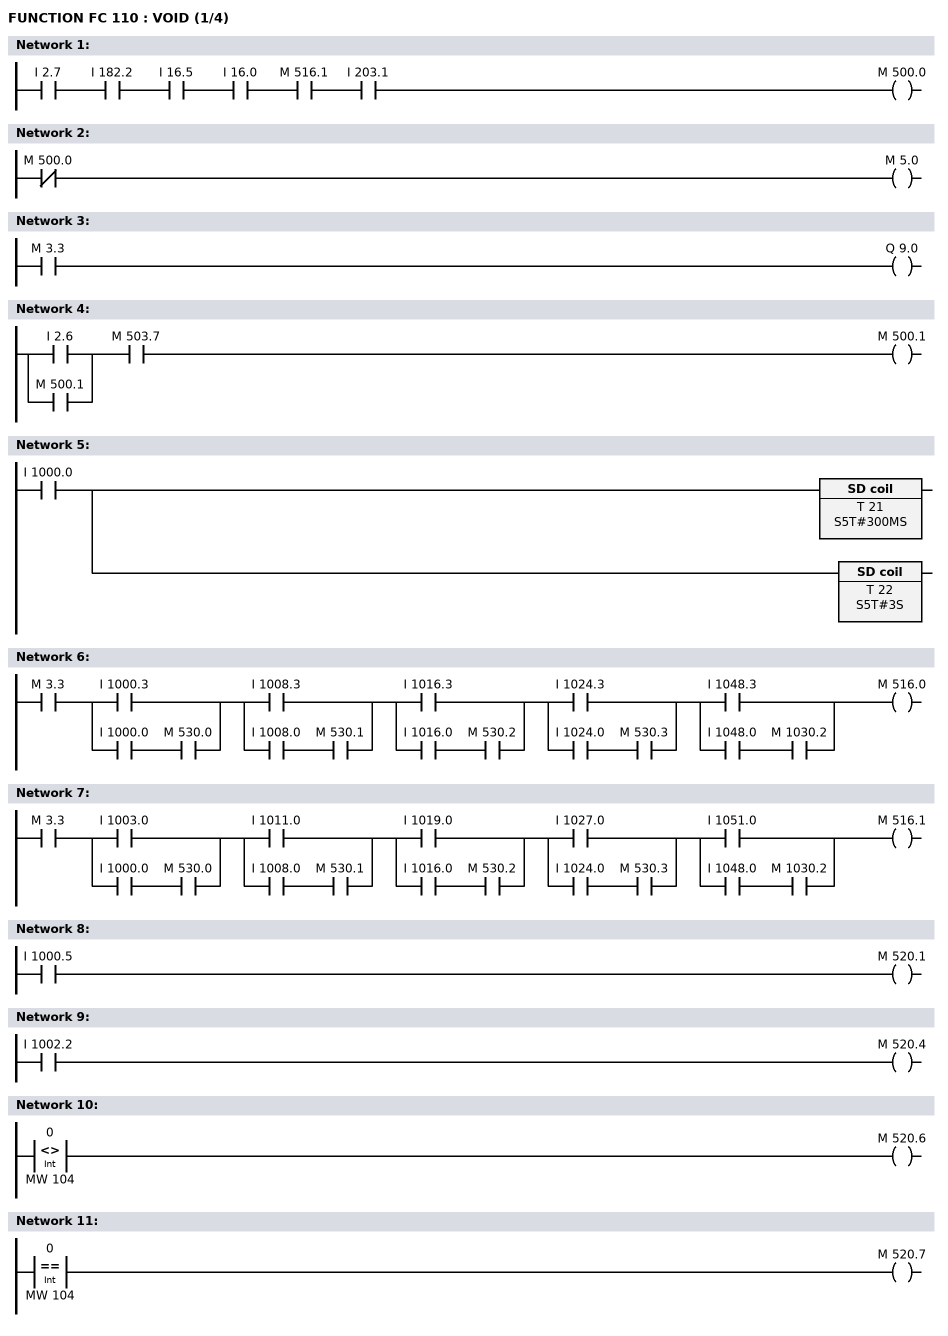

      A     I      2.7;
      A     I    182.2;
      A     I     16.5;
      A     I     16.0;
      A     M    516.1;
      A     I    203.1;
      =     M    500.0;
NETWORK
TITLE =

      AN    M    500.0;
      =     M      5.0;
NETWORK
TITLE =

      A     M      3.3;
      =     Q      9.0;
NETWORK
TITLE =

      A(    ;
      O     I      2.6;
      O     M    500.1;
      )     ;
      A     M    503.7;
      =     M    500.1;
NETWORK
TITLE =

      A     I   1000.0;
      L     S5T#300MS;
      SD    T     21;
      L     S5T#3S;
      SD    T     22;
NETWORK
TITLE =

      A     M      3.3;
      A(    ;
      O     I   1000.3;
      O     ;
      A     I   1000.0;
      A     M    530.0;
      )     ;
      A(    ;
      O     I   1008.3;
      O     ;
      A     I   1008.0;
      A     M    530.1;
      )     ;
      A(    ;
      O     I   1016.3;
      O     ;
      A     I   1016.0;
      A     M    530.2;
      )     ;
      A(    ;
      O     I   1024.3;
      O     ;
      A     I   1024.0;
      A     M    530.3;
      )     ;
      A(    ;
      O     I   1048.3;
      O     ;
      A     I   1048.0;
      A     M   1030.2;
      )     ;
      =     M    516.0;
NETWORK
TITLE =

      A     M      3.3;
      A(    ;
      O     I   1003.0;
      O     ;
      A     I   1000.0;
      A     M    530.0;
      )     ;
      A(    ;
      O     I   1011.0;
      O     ;
      A     I   1008.0;
      A     M    530.1;
      )     ;
      A(    ;
      O     I   1019.0;
      O     ;
      A     I   1016.0;
      A     M    530.2;
      )     ;
      A(    ;
      O     I   1027.0;
      O     ;
      A     I   1024.0;
      A     M    530.3;
      )     ;
      A(    ;
      O     I   1051.0;
      O     ;
      A     I   1048.0;
      A     M   1030.2;
      )     ;
      =     M    516.1;
NETWORK
TITLE =

      A     I   1000.5;
      =     M    520.1;
NETWORK
TITLE =

      A     I   1002.2;
      =     M    520.4;
NETWORK
TITLE =

      L     0;
      L     MW   104;
      <>I   ;
      =     M    520.6;
NETWORK
TITLE =

      L     0;
      L     MW   104;
      ==I   ;
      =     M    520.7;
NETWORK
TITLE =
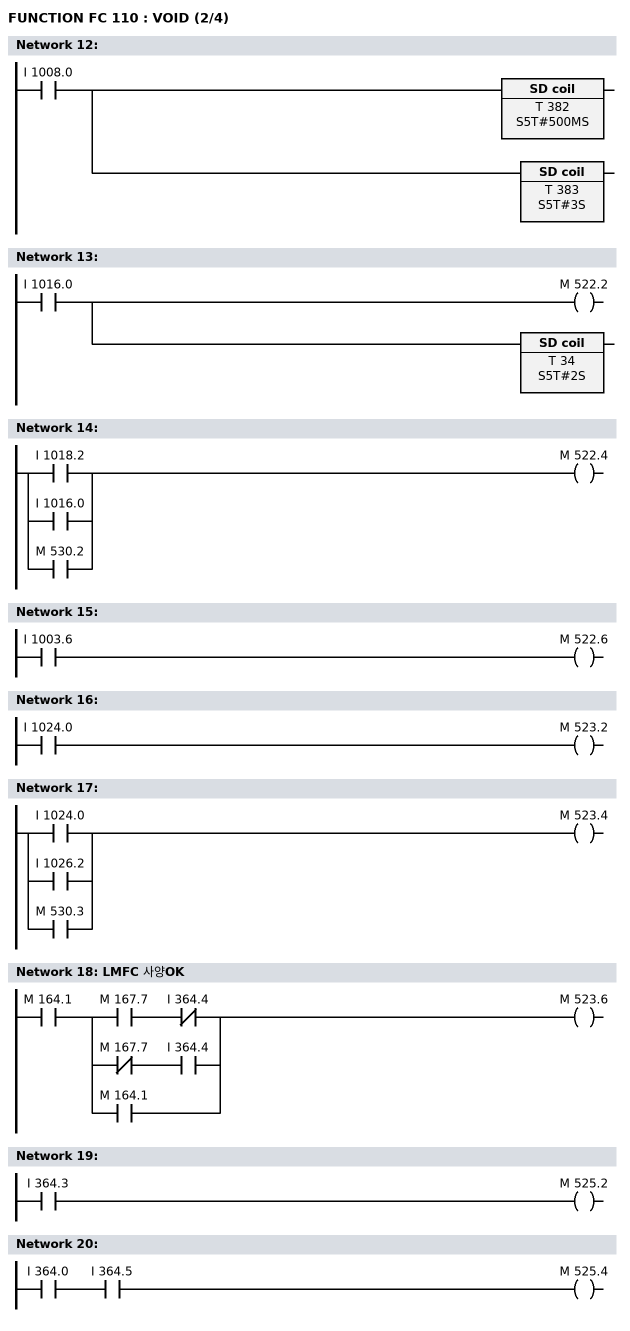

      A     I   1008.0;
      L     S5T#500MS;
      SD    T    382;
      L     S5T#3S;
      SD    T    383;
NETWORK
TITLE =

      A     I   1016.0;
      =     M    522.2;
      L     S5T#2S;
      SD    T     34;
NETWORK
TITLE =

      O     I   1018.2;
      O     I   1016.0;
      O     M    530.2;
      =     M    522.4;
NETWORK
TITLE =

      A     I   1003.6;
      =     M    522.6;
NETWORK
TITLE =

      A     I   1024.0;
      =     M    523.2;
NETWORK
TITLE =

      O     I   1024.0;
      O     I   1026.2;
      O     M    530.3;
      =     M    523.4;
NETWORK
TITLE =LMFC 사양OK

      A     M    164.1;
      A(    ;
      A     M    167.7;
      AN    I    364.4;
      O     ;
      AN    M    167.7;
      A     I    364.4;
      O     M    164.1;
      )     ;
      =     M    523.6;
NETWORK
TITLE =

      A     I    364.3;
      =     M    525.2;
NETWORK
TITLE =

      A     I    364.0;
      A     I    364.5;
      =     M    525.4;
NETWORK
TITLE =
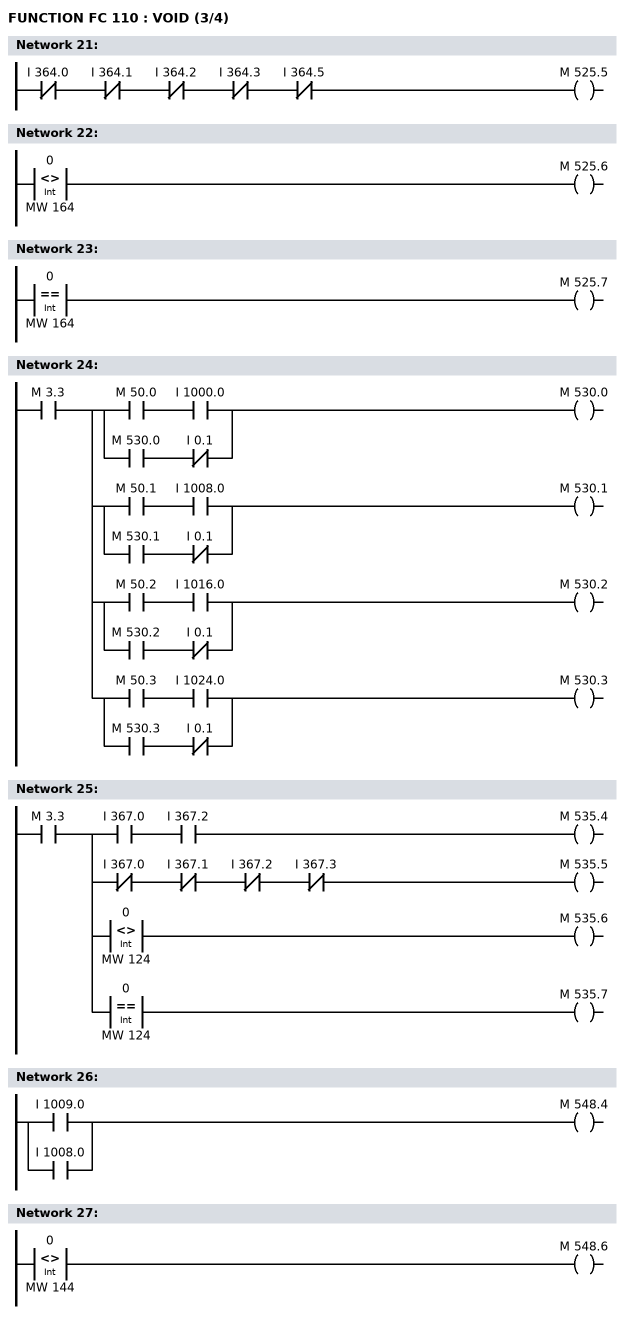

      AN    I    364.0;
      AN    I    364.1;
      AN    I    364.2;
      AN    I    364.3;
      AN    I    364.5;
      =     M    525.5;
NETWORK
TITLE =

      L     0;
      L     MW   164;
      <>I   ;
      =     M    525.6;
NETWORK
TITLE =

      L     0;
      L     MW   164;
      ==I   ;
      =     M    525.7;
NETWORK
TITLE =

      A     M      3.3;
      =     L      0.0;
      A     L      0.0;
      A(    ;
      A     M     50.0;
      A     I   1000.0;
      O     ;
      A     M    530.0;
      AN    I      0.1;
      )     ;
      =     M    530.0;
      A     L      0.0;
      A(    ;
      A     M     50.1;
      A     I   1008.0;
      O     ;
      A     M    530.1;
      AN    I      0.1;
      )     ;
      =     M    530.1;
      A     L      0.0;
      A(    ;
      A     M     50.2;
      A     I   1016.0;
      O     ;
      A     M    530.2;
      AN    I      0.1;
      )     ;
      =     M    530.2;
      A     L      0.0;
      A(    ;
      A     M     50.3;
      A     I   1024.0;
      O     ;
      A     M    530.3;
      AN    I      0.1;
      )     ;
      =     M    530.3;
NETWORK
TITLE =

      A     M      3.3;
      =     L      0.0;
      A     L      0.0;
      A     I    367.0;
      A     I    367.2;
      =     M    535.4;
      A     L      0.0;
      AN    I    367.0;
      AN    I    367.1;
      AN    I    367.2;
      AN    I    367.3;
      =     M    535.5;
      A     L      0.0;
      A(    ;
      L     0;
      L     MW   124;
      <>I   ;
      )     ;
      =     M    535.6;
      A     L      0.0;
      A(    ;
      L     0;
      L     MW   124;
      ==I   ;
      )     ;
      =     M    535.7;
NETWORK
TITLE =

      O     I   1009.0;
      O     I   1008.0;
      =     M    548.4;
NETWORK
TITLE =

      L     0;
      L     MW   144;
      <>I   ;
      =     M    548.6;
NETWORK
TITLE =
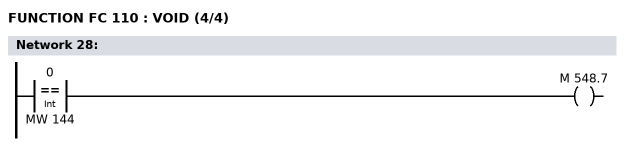

      L     0;
      L     MW   144;
      ==I   ;
      =     M    548.7;
END_FUNCTION

FUNCTION_BLOCK FB 111
TITLE =
VERSION : 0.1


VAR
  S700_1_TL_LATCH_ERR : FB 424;	//S700_1_TL_LATCH_ERR
  S700_1_TL_PIN_ERR : FB 424;	//S700_1_TL_PIN_ERR
  S700_1_LM_PIN_ERR : FB 424;	//S700_1_LM_PIN_ERR
  S700_1_LM_LATCH_ERR : FB 424;	//S700_1_LM_LATCH_ERR
END_VAR
BEGIN
NETWORK
TITLE =
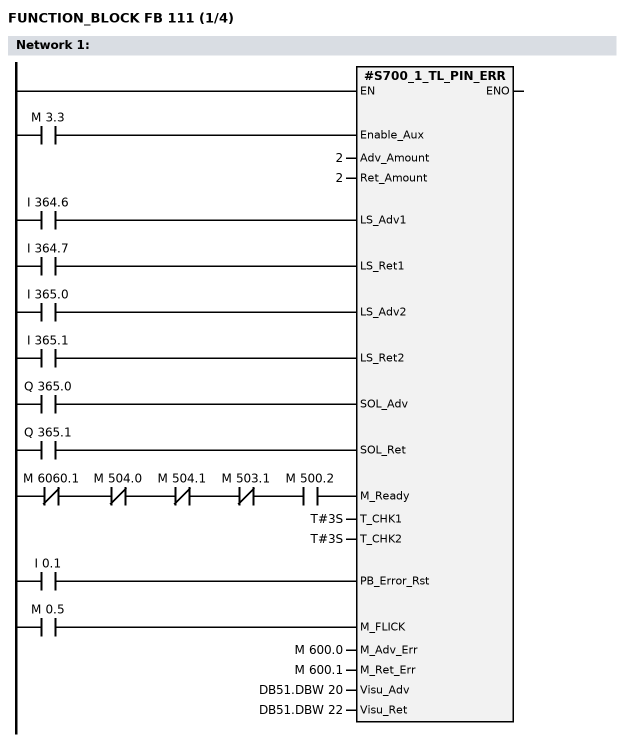

      A     M      3.3;
      =     L      0.0;
      BLD   103;
      A     I    364.6;
      =     L      0.1;
      BLD   103;
      A     I    364.7;
      =     L      0.2;
      BLD   103;
      A     I    365.0;
      =     L      0.3;
      BLD   103;
      A     I    365.1;
      =     L      0.4;
      BLD   103;
      A     Q    365.0;
      =     L      1.1;
      BLD   103;
      A     Q    365.1;
      =     L      1.2;
      BLD   103;
      AN    M   6060.1;
      AN    M    504.0;
      AN    M    504.1;
      AN    M    503.1;
      A     M    500.2;
      =     L      1.3;
      BLD   103;
      A     I      0.1;
      =     L      1.5;
      BLD   103;
      A     M      0.5;
      =     L      1.6;
      BLD   103;
      CALL #S700_1_TL_PIN_ERR (
           Enable_Aux               := L      0.0,
           Adv_Amount               := 2,
           Ret_Amount               := 2,
           LS_Adv1                  := L      0.1,
           LS_Ret1                  := L      0.2,
           LS_Adv2                  := L      0.3,
           LS_Ret2                  := L      0.4,
           SOL_Adv                  := L      1.1,
           SOL_Ret                  := L      1.2,
           M_Ready                  := L      1.3,
           T_CHK1                   := T#3S,
           T_CHK2                   := T#3S,
           PB_Error_Rst             := L      1.5,
           M_FLICK                  := L      1.6,
           M_Adv_Err                := M    600.0,
           M_Ret_Err                := M    600.1,
           Visu_Adv                 := DB51.DBW   20,
           Visu_Ret                 := DB51.DBW   22);
      NOP   0;
NETWORK
TITLE =
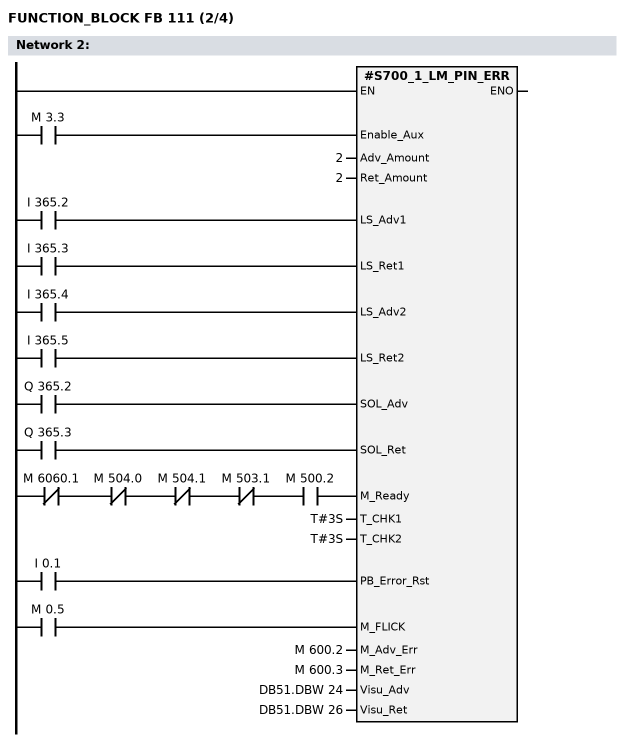

      A     M      3.3;
      =     L      0.0;
      BLD   103;
      A     I    365.2;
      =     L      0.1;
      BLD   103;
      A     I    365.3;
      =     L      0.2;
      BLD   103;
      A     I    365.4;
      =     L      0.3;
      BLD   103;
      A     I    365.5;
      =     L      0.4;
      BLD   103;
      A     Q    365.2;
      =     L      1.1;
      BLD   103;
      A     Q    365.3;
      =     L      1.2;
      BLD   103;
      AN    M   6060.1;
      AN    M    504.0;
      AN    M    504.1;
      AN    M    503.1;
      A     M    500.2;
      =     L      1.3;
      BLD   103;
      A     I      0.1;
      =     L      1.5;
      BLD   103;
      A     M      0.5;
      =     L      1.6;
      BLD   103;
      CALL #S700_1_LM_PIN_ERR (
           Enable_Aux               := L      0.0,
           Adv_Amount               := 2,
           Ret_Amount               := 2,
           LS_Adv1                  := L      0.1,
           LS_Ret1                  := L      0.2,
           LS_Adv2                  := L      0.3,
           LS_Ret2                  := L      0.4,
           SOL_Adv                  := L      1.1,
           SOL_Ret                  := L      1.2,
           M_Ready                  := L      1.3,
           T_CHK1                   := T#3S,
           T_CHK2                   := T#3S,
           PB_Error_Rst             := L      1.5,
           M_FLICK                  := L      1.6,
           M_Adv_Err                := M    600.2,
           M_Ret_Err                := M    600.3,
           Visu_Adv                 := DB51.DBW   24,
           Visu_Ret                 := DB51.DBW   26);
      NOP   0;
NETWORK
TITLE =
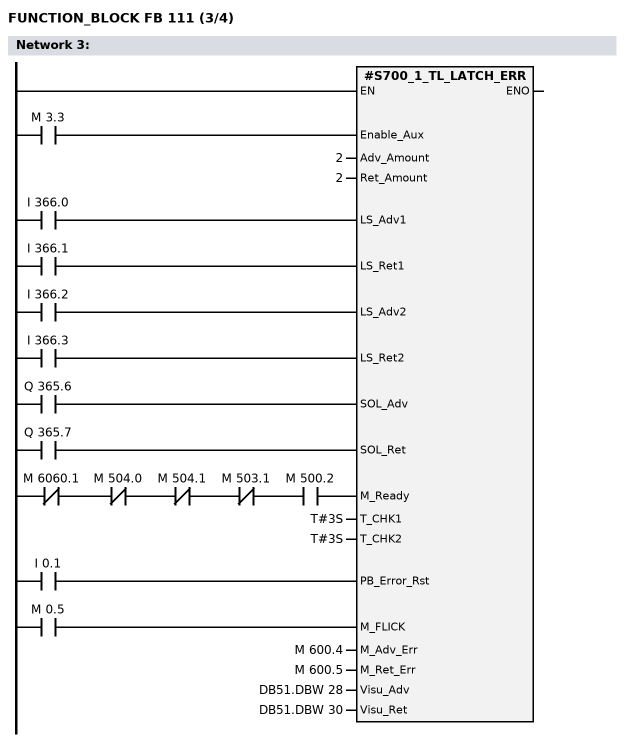

      A     M      3.3;
      =     L      0.0;
      BLD   103;
      A     I    366.0;
      =     L      0.1;
      BLD   103;
      A     I    366.1;
      =     L      0.2;
      BLD   103;
      A     I    366.2;
      =     L      0.3;
      BLD   103;
      A     I    366.3;
      =     L      0.4;
      BLD   103;
      A     Q    365.6;
      =     L      1.1;
      BLD   103;
      A     Q    365.7;
      =     L      1.2;
      BLD   103;
      AN    M   6060.1;
      AN    M    504.0;
      AN    M    504.1;
      AN    M    503.1;
      A     M    500.2;
      =     L      1.3;
      BLD   103;
      A     I      0.1;
      =     L      1.5;
      BLD   103;
      A     M      0.5;
      =     L      1.6;
      BLD   103;
      CALL #S700_1_TL_LATCH_ERR (
           Enable_Aux               := L      0.0,
           Adv_Amount               := 2,
           Ret_Amount               := 2,
           LS_Adv1                  := L      0.1,
           LS_Ret1                  := L      0.2,
           LS_Adv2                  := L      0.3,
           LS_Ret2                  := L      0.4,
           SOL_Adv                  := L      1.1,
           SOL_Ret                  := L      1.2,
           M_Ready                  := L      1.3,
           T_CHK1                   := T#3S,
           T_CHK2                   := T#3S,
           PB_Error_Rst             := L      1.5,
           M_FLICK                  := L      1.6,
           M_Adv_Err                := M    600.4,
           M_Ret_Err                := M    600.5,
           Visu_Adv                 := DB51.DBW   28,
           Visu_Ret                 := DB51.DBW   30);
      NOP   0;
NETWORK
TITLE =
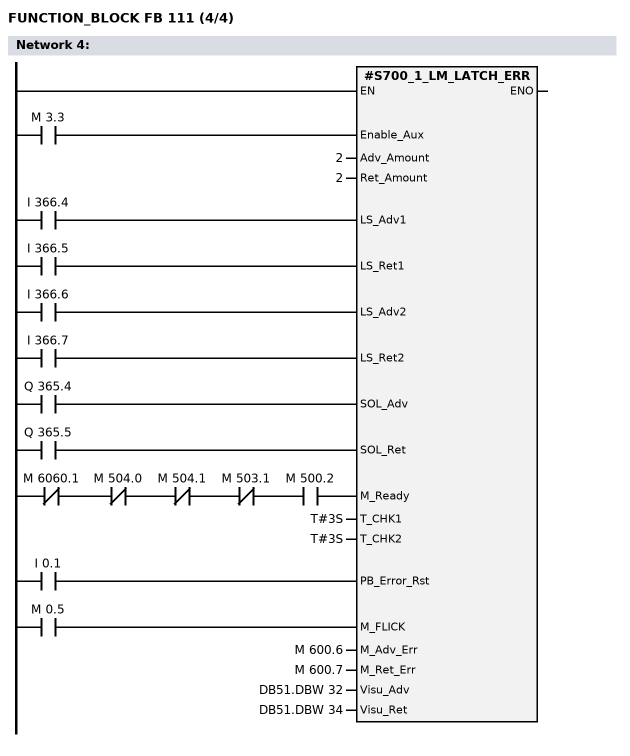

      A     M      3.3;
      =     L      0.0;
      BLD   103;
      A     I    366.4;
      =     L      0.1;
      BLD   103;
      A     I    366.5;
      =     L      0.2;
      BLD   103;
      A     I    366.6;
      =     L      0.3;
      BLD   103;
      A     I    366.7;
      =     L      0.4;
      BLD   103;
      A     Q    365.4;
      =     L      1.1;
      BLD   103;
      A     Q    365.5;
      =     L      1.2;
      BLD   103;
      AN    M   6060.1;
      AN    M    504.0;
      AN    M    504.1;
      AN    M    503.1;
      A     M    500.2;
      =     L      1.3;
      BLD   103;
      A     I      0.1;
      =     L      1.5;
      BLD   103;
      A     M      0.5;
      =     L      1.6;
      BLD   103;
      CALL #S700_1_LM_LATCH_ERR (
           Enable_Aux               := L      0.0,
           Adv_Amount               := 2,
           Ret_Amount               := 2,
           LS_Adv1                  := L      0.1,
           LS_Ret1                  := L      0.2,
           LS_Adv2                  := L      0.3,
           LS_Ret2                  := L      0.4,
           SOL_Adv                  := L      1.1,
           SOL_Ret                  := L      1.2,
           M_Ready                  := L      1.3,
           T_CHK1                   := T#3S,
           T_CHK2                   := T#3S,
           PB_Error_Rst             := L      1.5,
           M_FLICK                  := L      1.6,
           M_Adv_Err                := M    600.6,
           M_Ret_Err                := M    600.7,
           Visu_Adv                 := DB51.DBW   32,
           Visu_Ret                 := DB51.DBW   34);
      NOP   0;
END_FUNCTION_BLOCK

DATA_BLOCK DB 111
TITLE =
VERSION : 0.0

 FB 111
BEGIN
   S700_1_TL_LATCH_ERR.Enable_Aux := FALSE;
   S700_1_TL_LATCH_ERR.Adv_Amount := 0;
   S700_1_TL_LATCH_ERR.Ret_Amount := 0;
   S700_1_TL_LATCH_ERR.LS_Adv1 := FALSE;
   S700_1_TL_LATCH_ERR.LS_Ret1 := FALSE;
   S700_1_TL_LATCH_ERR.LS_Adv2 := FALSE;
   S700_1_TL_LATCH_ERR.LS_Ret2 := FALSE;
   S700_1_TL_LATCH_ERR.LS_Adv3 := FALSE;
   S700_1_TL_LATCH_ERR.LS_Ret3 := FALSE;
   S700_1_TL_LATCH_ERR.LS_Adv4 := FALSE;
   S700_1_TL_LATCH_ERR.LS_Ret4 := FALSE;
   S700_1_TL_LATCH_ERR.SOL_Adv := FALSE;
   S700_1_TL_LATCH_ERR.SOL_Ret := FALSE;
   S700_1_TL_LATCH_ERR.M_Ready := FALSE;
   S700_1_TL_LATCH_ERR.T_CHK1 := T#0MS;
   S700_1_TL_LATCH_ERR.T_CHK2 := T#0MS;
   S700_1_TL_LATCH_ERR.PB_Lamp_CHK := FALSE;
   S700_1_TL_LATCH_ERR.PB_Error_Rst := FALSE;
   S700_1_TL_LATCH_ERR.M_FLICK := FALSE;
   S700_1_TL_LATCH_ERR.M_Adv_Err := FALSE;
   S700_1_TL_LATCH_ERR.M_Ret_Err := FALSE;
   S700_1_TL_LATCH_ERR.LP_Adv := FALSE;
   S700_1_TL_LATCH_ERR.LP_Ret := FALSE;
   S700_1_TL_LATCH_ERR.Visu_Adv := W#16#0;
   S700_1_TL_LATCH_ERR.Visu_Ret := W#16#0;
   S700_1_TL_LATCH_ERR.Error_T1.IN := FALSE;
   S700_1_TL_LATCH_ERR.Error_T1.PT := T#0MS;
   S700_1_TL_LATCH_ERR.Error_T1.Q := FALSE;
   S700_1_TL_LATCH_ERR.Error_T1.ET := T#0MS;
   S700_1_TL_LATCH_ERR.Error_T1.STATE := B#16#0;
   S700_1_TL_LATCH_ERR.Error_T1.STIME := T#0MS;
   S700_1_TL_LATCH_ERR.Error_T1.ATIME := T#0MS;
   S700_1_TL_LATCH_ERR.Error_T2.IN := FALSE;
   S700_1_TL_LATCH_ERR.Error_T2.PT := T#0MS;
   S700_1_TL_LATCH_ERR.Error_T2.Q := FALSE;
   S700_1_TL_LATCH_ERR.Error_T2.ET := T#0MS;
   S700_1_TL_LATCH_ERR.Error_T2.STATE := B#16#0;
   S700_1_TL_LATCH_ERR.Error_T2.STIME := T#0MS;
   S700_1_TL_LATCH_ERR.Error_T2.ATIME := T#0MS;
   S700_1_TL_LATCH_ERR.CHK_Aux1 := FALSE;
   S700_1_TL_LATCH_ERR.CHK_Aux2 := FALSE;
   S700_1_TL_LATCH_ERR.Error_T1_DN := FALSE;
   S700_1_TL_LATCH_ERR.Error_T2_DN := FALSE;
   S700_1_TL_LATCH_ERR.Adv_Memo := FALSE;
   S700_1_TL_LATCH_ERR.Visu_Adv_Arr[0] := FALSE;
   S700_1_TL_LATCH_ERR.Visu_Adv_Arr[1] := FALSE;
   S700_1_TL_LATCH_ERR.Visu_Adv_Arr[2] := FALSE;
   S700_1_TL_LATCH_ERR.Visu_Adv_Arr[3] := FALSE;
   S700_1_TL_LATCH_ERR.Visu_Adv_Arr[4] := FALSE;
   S700_1_TL_LATCH_ERR.Visu_Adv_Arr[5] := FALSE;
   S700_1_TL_LATCH_ERR.Visu_Adv_Arr[6] := FALSE;
   S700_1_TL_LATCH_ERR.Visu_Adv_Arr[7] := FALSE;
   S700_1_TL_LATCH_ERR.Visu_Adv_Arr[8] := FALSE;
   S700_1_TL_LATCH_ERR.Visu_Adv_Arr[9] := FALSE;
   S700_1_TL_LATCH_ERR.Visu_Adv_Arr[10] := FALSE;
   S700_1_TL_LATCH_ERR.Visu_Adv_Arr[11] := FALSE;
   S700_1_TL_LATCH_ERR.Visu_Adv_Arr[12] := FALSE;
   S700_1_TL_LATCH_ERR.Visu_Adv_Arr[13] := FALSE;
   S700_1_TL_LATCH_ERR.Visu_Adv_Arr[14] := FALSE;
   S700_1_TL_LATCH_ERR.Visu_Adv_Arr[15] := FALSE;
   S700_1_TL_LATCH_ERR.Visu_Ret_Arr[0] := FALSE;
   S700_1_TL_LATCH_ERR.Visu_Ret_Arr[1] := FALSE;
   S700_1_TL_LATCH_ERR.Visu_Ret_Arr[2] := FALSE;
   S700_1_TL_LATCH_ERR.Visu_Ret_Arr[3] := FALSE;
   S700_1_TL_LATCH_ERR.Visu_Ret_Arr[4] := FALSE;
   S700_1_TL_LATCH_ERR.Visu_Ret_Arr[5] := FALSE;
   S700_1_TL_LATCH_ERR.Visu_Ret_Arr[6] := FALSE;
   S700_1_TL_LATCH_ERR.Visu_Ret_Arr[7] := FALSE;
   S700_1_TL_LATCH_ERR.Visu_Ret_Arr[8] := FALSE;
   S700_1_TL_LATCH_ERR.Visu_Ret_Arr[9] := FALSE;
   S700_1_TL_LATCH_ERR.Visu_Ret_Arr[10] := FALSE;
   S700_1_TL_LATCH_ERR.Visu_Ret_Arr[11] := FALSE;
   S700_1_TL_LATCH_ERR.Visu_Ret_Arr[12] := FALSE;
   S700_1_TL_LATCH_ERR.Visu_Ret_Arr[13] := FALSE;
   S700_1_TL_LATCH_ERR.Visu_Ret_Arr[14] := FALSE;
   S700_1_TL_LATCH_ERR.Visu_Ret_Arr[15] := FALSE;
   S700_1_TL_LATCH_ERR.BLK_Move_Ret := 0;
   S700_1_TL_LATCH_ERR.Enable := FALSE;
   S700_1_TL_LATCH_ERR.Adv_End := FALSE;
   S700_1_TL_LATCH_ERR.Ret_End := FALSE;
   S700_1_TL_PIN_ERR.Enable_Aux := FALSE;
   S700_1_TL_PIN_ERR.Adv_Amount := 0;
   S700_1_TL_PIN_ERR.Ret_Amount := 0;
   S700_1_TL_PIN_ERR.LS_Adv1 := FALSE;
   S700_1_TL_PIN_ERR.LS_Ret1 := FALSE;
   S700_1_TL_PIN_ERR.LS_Adv2 := FALSE;
   S700_1_TL_PIN_ERR.LS_Ret2 := FALSE;
   S700_1_TL_PIN_ERR.LS_Adv3 := FALSE;
   S700_1_TL_PIN_ERR.LS_Ret3 := FALSE;
   S700_1_TL_PIN_ERR.LS_Adv4 := FALSE;
   S700_1_TL_PIN_ERR.LS_Ret4 := FALSE;
   S700_1_TL_PIN_ERR.SOL_Adv := FALSE;
   S700_1_TL_PIN_ERR.SOL_Ret := FALSE;
   S700_1_TL_PIN_ERR.M_Ready := FALSE;
   S700_1_TL_PIN_ERR.T_CHK1 := T#0MS;
   S700_1_TL_PIN_ERR.T_CHK2 := T#0MS;
   S700_1_TL_PIN_ERR.PB_Lamp_CHK := FALSE;
   S700_1_TL_PIN_ERR.PB_Error_Rst := FALSE;
   S700_1_TL_PIN_ERR.M_FLICK := FALSE;
   S700_1_TL_PIN_ERR.M_Adv_Err := FALSE;
   S700_1_TL_PIN_ERR.M_Ret_Err := FALSE;
   S700_1_TL_PIN_ERR.LP_Adv := FALSE;
   S700_1_TL_PIN_ERR.LP_Ret := FALSE;
   S700_1_TL_PIN_ERR.Visu_Adv := W#16#0;
   S700_1_TL_PIN_ERR.Visu_Ret := W#16#0;
   S700_1_TL_PIN_ERR.Error_T1.IN := FALSE;
   S700_1_TL_PIN_ERR.Error_T1.PT := T#0MS;
   S700_1_TL_PIN_ERR.Error_T1.Q := FALSE;
   S700_1_TL_PIN_ERR.Error_T1.ET := T#0MS;
   S700_1_TL_PIN_ERR.Error_T1.STATE := B#16#0;
   S700_1_TL_PIN_ERR.Error_T1.STIME := T#0MS;
   S700_1_TL_PIN_ERR.Error_T1.ATIME := T#0MS;
   S700_1_TL_PIN_ERR.Error_T2.IN := FALSE;
   S700_1_TL_PIN_ERR.Error_T2.PT := T#0MS;
   S700_1_TL_PIN_ERR.Error_T2.Q := FALSE;
   S700_1_TL_PIN_ERR.Error_T2.ET := T#0MS;
   S700_1_TL_PIN_ERR.Error_T2.STATE := B#16#0;
   S700_1_TL_PIN_ERR.Error_T2.STIME := T#0MS;
   S700_1_TL_PIN_ERR.Error_T2.ATIME := T#0MS;
   S700_1_TL_PIN_ERR.CHK_Aux1 := FALSE;
   S700_1_TL_PIN_ERR.CHK_Aux2 := FALSE;
   S700_1_TL_PIN_ERR.Error_T1_DN := FALSE;
   S700_1_TL_PIN_ERR.Error_T2_DN := FALSE;
   S700_1_TL_PIN_ERR.Adv_Memo := FALSE;
   S700_1_TL_PIN_ERR.Visu_Adv_Arr[0] := FALSE;
   S700_1_TL_PIN_ERR.Visu_Adv_Arr[1] := FALSE;
   S700_1_TL_PIN_ERR.Visu_Adv_Arr[2] := FALSE;
   S700_1_TL_PIN_ERR.Visu_Adv_Arr[3] := FALSE;
   S700_1_TL_PIN_ERR.Visu_Adv_Arr[4] := FALSE;
   S700_1_TL_PIN_ERR.Visu_Adv_Arr[5] := FALSE;
   S700_1_TL_PIN_ERR.Visu_Adv_Arr[6] := FALSE;
   S700_1_TL_PIN_ERR.Visu_Adv_Arr[7] := FALSE;
   S700_1_TL_PIN_ERR.Visu_Adv_Arr[8] := FALSE;
   S700_1_TL_PIN_ERR.Visu_Adv_Arr[9] := FALSE;
   S700_1_TL_PIN_ERR.Visu_Adv_Arr[10] := FALSE;
   S700_1_TL_PIN_ERR.Visu_Adv_Arr[11] := FALSE;
   S700_1_TL_PIN_ERR.Visu_Adv_Arr[12] := FALSE;
   S700_1_TL_PIN_ERR.Visu_Adv_Arr[13] := FALSE;
   S700_1_TL_PIN_ERR.Visu_Adv_Arr[14] := FALSE;
   S700_1_TL_PIN_ERR.Visu_Adv_Arr[15] := FALSE;
   S700_1_TL_PIN_ERR.Visu_Ret_Arr[0] := FALSE;
   S700_1_TL_PIN_ERR.Visu_Ret_Arr[1] := FALSE;
   S700_1_TL_PIN_ERR.Visu_Ret_Arr[2] := FALSE;
   S700_1_TL_PIN_ERR.Visu_Ret_Arr[3] := FALSE;
   S700_1_TL_PIN_ERR.Visu_Ret_Arr[4] := FALSE;
   S700_1_TL_PIN_ERR.Visu_Ret_Arr[5] := FALSE;
   S700_1_TL_PIN_ERR.Visu_Ret_Arr[6] := FALSE;
   S700_1_TL_PIN_ERR.Visu_Ret_Arr[7] := FALSE;
   S700_1_TL_PIN_ERR.Visu_Ret_Arr[8] := FALSE;
   S700_1_TL_PIN_ERR.Visu_Ret_Arr[9] := FALSE;
   S700_1_TL_PIN_ERR.Visu_Ret_Arr[10] := FALSE;
   S700_1_TL_PIN_ERR.Visu_Ret_Arr[11] := FALSE;
   S700_1_TL_PIN_ERR.Visu_Ret_Arr[12] := FALSE;
   S700_1_TL_PIN_ERR.Visu_Ret_Arr[13] := FALSE;
   S700_1_TL_PIN_ERR.Visu_Ret_Arr[14] := FALSE;
   S700_1_TL_PIN_ERR.Visu_Ret_Arr[15] := FALSE;
   S700_1_TL_PIN_ERR.BLK_Move_Ret := 0;
   S700_1_TL_PIN_ERR.Enable := FALSE;
   S700_1_TL_PIN_ERR.Adv_End := FALSE;
   S700_1_TL_PIN_ERR.Ret_End := FALSE;
   S700_1_LM_PIN_ERR.Enable_Aux := FALSE;
   S700_1_LM_PIN_ERR.Adv_Amount := 0;
   S700_1_LM_PIN_ERR.Ret_Amount := 0;
   S700_1_LM_PIN_ERR.LS_Adv1 := FALSE;
   S700_1_LM_PIN_ERR.LS_Ret1 := FALSE;
   S700_1_LM_PIN_ERR.LS_Adv2 := FALSE;
   S700_1_LM_PIN_ERR.LS_Ret2 := FALSE;
   S700_1_LM_PIN_ERR.LS_Adv3 := FALSE;
   S700_1_LM_PIN_ERR.LS_Ret3 := FALSE;
   S700_1_LM_PIN_ERR.LS_Adv4 := FALSE;
   S700_1_LM_PIN_ERR.LS_Ret4 := FALSE;
   S700_1_LM_PIN_ERR.SOL_Adv := FALSE;
   S700_1_LM_PIN_ERR.SOL_Ret := FALSE;
   S700_1_LM_PIN_ERR.M_Ready := FALSE;
   S700_1_LM_PIN_ERR.T_CHK1 := T#0MS;
   S700_1_LM_PIN_ERR.T_CHK2 := T#0MS;
   S700_1_LM_PIN_ERR.PB_Lamp_CHK := FALSE;
   S700_1_LM_PIN_ERR.PB_Error_Rst := FALSE;
   S700_1_LM_PIN_ERR.M_FLICK := FALSE;
   S700_1_LM_PIN_ERR.M_Adv_Err := FALSE;
   S700_1_LM_PIN_ERR.M_Ret_Err := FALSE;
   S700_1_LM_PIN_ERR.LP_Adv := FALSE;
   S700_1_LM_PIN_ERR.LP_Ret := FALSE;
   S700_1_LM_PIN_ERR.Visu_Adv := W#16#0;
   S700_1_LM_PIN_ERR.Visu_Ret := W#16#0;
   S700_1_LM_PIN_ERR.Error_T1.IN := FALSE;
   S700_1_LM_PIN_ERR.Error_T1.PT := T#0MS;
   S700_1_LM_PIN_ERR.Error_T1.Q := FALSE;
   S700_1_LM_PIN_ERR.Error_T1.ET := T#0MS;
   S700_1_LM_PIN_ERR.Error_T1.STATE := B#16#0;
   S700_1_LM_PIN_ERR.Error_T1.STIME := T#0MS;
   S700_1_LM_PIN_ERR.Error_T1.ATIME := T#0MS;
   S700_1_LM_PIN_ERR.Error_T2.IN := FALSE;
   S700_1_LM_PIN_ERR.Error_T2.PT := T#0MS;
   S700_1_LM_PIN_ERR.Error_T2.Q := FALSE;
   S700_1_LM_PIN_ERR.Error_T2.ET := T#0MS;
   S700_1_LM_PIN_ERR.Error_T2.STATE := B#16#0;
   S700_1_LM_PIN_ERR.Error_T2.STIME := T#0MS;
   S700_1_LM_PIN_ERR.Error_T2.ATIME := T#0MS;
   S700_1_LM_PIN_ERR.CHK_Aux1 := FALSE;
   S700_1_LM_PIN_ERR.CHK_Aux2 := FALSE;
   S700_1_LM_PIN_ERR.Error_T1_DN := FALSE;
   S700_1_LM_PIN_ERR.Error_T2_DN := FALSE;
   S700_1_LM_PIN_ERR.Adv_Memo := FALSE;
   S700_1_LM_PIN_ERR.Visu_Adv_Arr[0] := FALSE;
   S700_1_LM_PIN_ERR.Visu_Adv_Arr[1] := FALSE;
   S700_1_LM_PIN_ERR.Visu_Adv_Arr[2] := FALSE;
   S700_1_LM_PIN_ERR.Visu_Adv_Arr[3] := FALSE;
   S700_1_LM_PIN_ERR.Visu_Adv_Arr[4] := FALSE;
   S700_1_LM_PIN_ERR.Visu_Adv_Arr[5] := FALSE;
   S700_1_LM_PIN_ERR.Visu_Adv_Arr[6] := FALSE;
   S700_1_LM_PIN_ERR.Visu_Adv_Arr[7] := FALSE;
   S700_1_LM_PIN_ERR.Visu_Adv_Arr[8] := FALSE;
   S700_1_LM_PIN_ERR.Visu_Adv_Arr[9] := FALSE;
   S700_1_LM_PIN_ERR.Visu_Adv_Arr[10] := FALSE;
   S700_1_LM_PIN_ERR.Visu_Adv_Arr[11] := FALSE;
   S700_1_LM_PIN_ERR.Visu_Adv_Arr[12] := FALSE;
   S700_1_LM_PIN_ERR.Visu_Adv_Arr[13] := FALSE;
   S700_1_LM_PIN_ERR.Visu_Adv_Arr[14] := FALSE;
   S700_1_LM_PIN_ERR.Visu_Adv_Arr[15] := FALSE;
   S700_1_LM_PIN_ERR.Visu_Ret_Arr[0] := FALSE;
   S700_1_LM_PIN_ERR.Visu_Ret_Arr[1] := FALSE;
   S700_1_LM_PIN_ERR.Visu_Ret_Arr[2] := FALSE;
   S700_1_LM_PIN_ERR.Visu_Ret_Arr[3] := FALSE;
   S700_1_LM_PIN_ERR.Visu_Ret_Arr[4] := FALSE;
   S700_1_LM_PIN_ERR.Visu_Ret_Arr[5] := FALSE;
   S700_1_LM_PIN_ERR.Visu_Ret_Arr[6] := FALSE;
   S700_1_LM_PIN_ERR.Visu_Ret_Arr[7] := FALSE;
   S700_1_LM_PIN_ERR.Visu_Ret_Arr[8] := FALSE;
   S700_1_LM_PIN_ERR.Visu_Ret_Arr[9] := FALSE;
   S700_1_LM_PIN_ERR.Visu_Ret_Arr[10] := FALSE;
   S700_1_LM_PIN_ERR.Visu_Ret_Arr[11] := FALSE;
   S700_1_LM_PIN_ERR.Visu_Ret_Arr[12] := FALSE;
   S700_1_LM_PIN_ERR.Visu_Ret_Arr[13] := FALSE;
   S700_1_LM_PIN_ERR.Visu_Ret_Arr[14] := FALSE;
   S700_1_LM_PIN_ERR.Visu_Ret_Arr[15] := FALSE;
   S700_1_LM_PIN_ERR.BLK_Move_Ret := 0;
   S700_1_LM_PIN_ERR.Enable := FALSE;
   S700_1_LM_PIN_ERR.Adv_End := FALSE;
   S700_1_LM_PIN_ERR.Ret_End := FALSE;
   S700_1_LM_LATCH_ERR.Enable_Aux := FALSE;
   S700_1_LM_LATCH_ERR.Adv_Amount := 0;
   S700_1_LM_LATCH_ERR.Ret_Amount := 0;
   S700_1_LM_LATCH_ERR.LS_Adv1 := FALSE;
   S700_1_LM_LATCH_ERR.LS_Ret1 := FALSE;
   S700_1_LM_LATCH_ERR.LS_Adv2 := FALSE;
   S700_1_LM_LATCH_ERR.LS_Ret2 := FALSE;
   S700_1_LM_LATCH_ERR.LS_Adv3 := FALSE;
   S700_1_LM_LATCH_ERR.LS_Ret3 := FALSE;
   S700_1_LM_LATCH_ERR.LS_Adv4 := FALSE;
   S700_1_LM_LATCH_ERR.LS_Ret4 := FALSE;
   S700_1_LM_LATCH_ERR.SOL_Adv := FALSE;
   S700_1_LM_LATCH_ERR.SOL_Ret := FALSE;
   S700_1_LM_LATCH_ERR.M_Ready := FALSE;
   S700_1_LM_LATCH_ERR.T_CHK1 := T#0MS;
   S700_1_LM_LATCH_ERR.T_CHK2 := T#0MS;
   S700_1_LM_LATCH_ERR.PB_Lamp_CHK := FALSE;
   S700_1_LM_LATCH_ERR.PB_Error_Rst := FALSE;
   S700_1_LM_LATCH_ERR.M_FLICK := FALSE;
   S700_1_LM_LATCH_ERR.M_Adv_Err := FALSE;
   S700_1_LM_LATCH_ERR.M_Ret_Err := FALSE;
   S700_1_LM_LATCH_ERR.LP_Adv := FALSE;
   S700_1_LM_LATCH_ERR.LP_Ret := FALSE;
   S700_1_LM_LATCH_ERR.Visu_Adv := W#16#0;
   S700_1_LM_LATCH_ERR.Visu_Ret := W#16#0;
   S700_1_LM_LATCH_ERR.Error_T1.IN := FALSE;
   S700_1_LM_LATCH_ERR.Error_T1.PT := T#0MS;
   S700_1_LM_LATCH_ERR.Error_T1.Q := FALSE;
   S700_1_LM_LATCH_ERR.Error_T1.ET := T#0MS;
   S700_1_LM_LATCH_ERR.Error_T1.STATE := B#16#0;
   S700_1_LM_LATCH_ERR.Error_T1.STIME := T#0MS;
   S700_1_LM_LATCH_ERR.Error_T1.ATIME := T#0MS;
   S700_1_LM_LATCH_ERR.Error_T2.IN := FALSE;
   S700_1_LM_LATCH_ERR.Error_T2.PT := T#0MS;
   S700_1_LM_LATCH_ERR.Error_T2.Q := FALSE;
   S700_1_LM_LATCH_ERR.Error_T2.ET := T#0MS;
   S700_1_LM_LATCH_ERR.Error_T2.STATE := B#16#0;
   S700_1_LM_LATCH_ERR.Error_T2.STIME := T#0MS;
   S700_1_LM_LATCH_ERR.Error_T2.ATIME := T#0MS;
   S700_1_LM_LATCH_ERR.CHK_Aux1 := FALSE;
   S700_1_LM_LATCH_ERR.CHK_Aux2 := FALSE;
   S700_1_LM_LATCH_ERR.Error_T1_DN := FALSE;
   S700_1_LM_LATCH_ERR.Error_T2_DN := FALSE;
   S700_1_LM_LATCH_ERR.Adv_Memo := FALSE;
   S700_1_LM_LATCH_ERR.Visu_Adv_Arr[0] := FALSE;
   S700_1_LM_LATCH_ERR.Visu_Adv_Arr[1] := FALSE;
   S700_1_LM_LATCH_ERR.Visu_Adv_Arr[2] := FALSE;
   S700_1_LM_LATCH_ERR.Visu_Adv_Arr[3] := FALSE;
   S700_1_LM_LATCH_ERR.Visu_Adv_Arr[4] := FALSE;
   S700_1_LM_LATCH_ERR.Visu_Adv_Arr[5] := FALSE;
   S700_1_LM_LATCH_ERR.Visu_Adv_Arr[6] := FALSE;
   S700_1_LM_LATCH_ERR.Visu_Adv_Arr[7] := FALSE;
   S700_1_LM_LATCH_ERR.Visu_Adv_Arr[8] := FALSE;
   S700_1_LM_LATCH_ERR.Visu_Adv_Arr[9] := FALSE;
   S700_1_LM_LATCH_ERR.Visu_Adv_Arr[10] := FALSE;
   S700_1_LM_LATCH_ERR.Visu_Adv_Arr[11] := FALSE;
   S700_1_LM_LATCH_ERR.Visu_Adv_Arr[12] := FALSE;
   S700_1_LM_LATCH_ERR.Visu_Adv_Arr[13] := FALSE;
   S700_1_LM_LATCH_ERR.Visu_Adv_Arr[14] := FALSE;
   S700_1_LM_LATCH_ERR.Visu_Adv_Arr[15] := FALSE;
   S700_1_LM_LATCH_ERR.Visu_Ret_Arr[0] := FALSE;
   S700_1_LM_LATCH_ERR.Visu_Ret_Arr[1] := FALSE;
   S700_1_LM_LATCH_ERR.Visu_Ret_Arr[2] := FALSE;
   S700_1_LM_LATCH_ERR.Visu_Ret_Arr[3] := FALSE;
   S700_1_LM_LATCH_ERR.Visu_Ret_Arr[4] := FALSE;
   S700_1_LM_LATCH_ERR.Visu_Ret_Arr[5] := FALSE;
   S700_1_LM_LATCH_ERR.Visu_Ret_Arr[6] := FALSE;
   S700_1_LM_LATCH_ERR.Visu_Ret_Arr[7] := FALSE;
   S700_1_LM_LATCH_ERR.Visu_Ret_Arr[8] := FALSE;
   S700_1_LM_LATCH_ERR.Visu_Ret_Arr[9] := FALSE;
   S700_1_LM_LATCH_ERR.Visu_Ret_Arr[10] := FALSE;
   S700_1_LM_LATCH_ERR.Visu_Ret_Arr[11] := FALSE;
   S700_1_LM_LATCH_ERR.Visu_Ret_Arr[12] := FALSE;
   S700_1_LM_LATCH_ERR.Visu_Ret_Arr[13] := FALSE;
   S700_1_LM_LATCH_ERR.Visu_Ret_Arr[14] := FALSE;
   S700_1_LM_LATCH_ERR.Visu_Ret_Arr[15] := FALSE;
   S700_1_LM_LATCH_ERR.BLK_Move_Ret := 0;
   S700_1_LM_LATCH_ERR.Enable := FALSE;
   S700_1_LM_LATCH_ERR.Adv_End := FALSE;
   S700_1_LM_LATCH_ERR.Ret_End := FALSE;
END_DATA_BLOCK

FUNCTION FC 111 : VOID
TITLE =
VERSION : 0.1

BEGIN
NETWORK
TITLE =
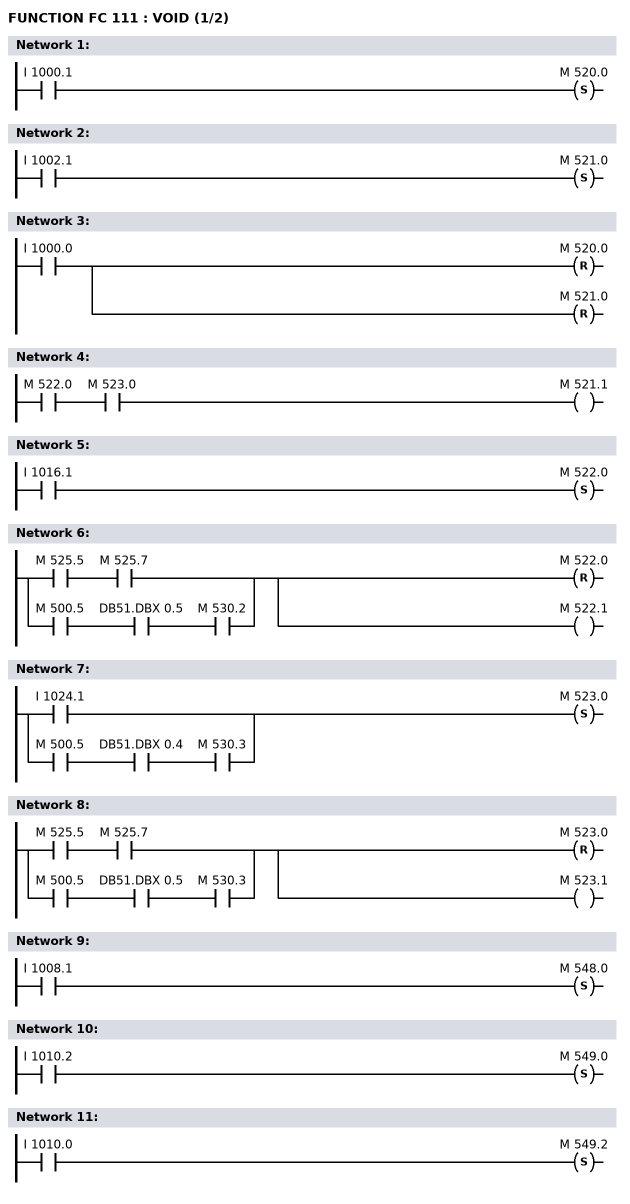

      A     I   1000.1;
      S     M    520.0;
NETWORK
TITLE =

      A     I   1002.1;
      S     M    521.0;
NETWORK
TITLE =

      A     I   1000.0;
      R     M    520.0;
      R     M    521.0;
NETWORK
TITLE =

      A     M    522.0;
      A     M    523.0;
      =     M    521.1;
NETWORK
TITLE =

      A     I   1016.1;
      S     M    522.0;
NETWORK
TITLE =

      A     M    525.5;
      A     M    525.7;
      O     ;
      A     M    500.5;
      A     DB51.DBX    0.5;
      A     M    530.2;
      R     M    522.0;
      =     M    522.1;
NETWORK
TITLE =

      O     I   1024.1;
      O     ;
      A     M    500.5;
      A     DB51.DBX    0.4;
      A     M    530.3;
      S     M    523.0;
NETWORK
TITLE =

      A     M    525.5;
      A     M    525.7;
      O     ;
      A     M    500.5;
      A     DB51.DBX    0.5;
      A     M    530.3;
      R     M    523.0;
      =     M    523.1;
NETWORK
TITLE =

      A     I   1008.1;
      S     M    548.0;
NETWORK
TITLE =

      A     I   1010.2;
      S     M    549.0;
NETWORK
TITLE =

      A     I   1010.0;
      S     M    549.2;
NETWORK
TITLE =
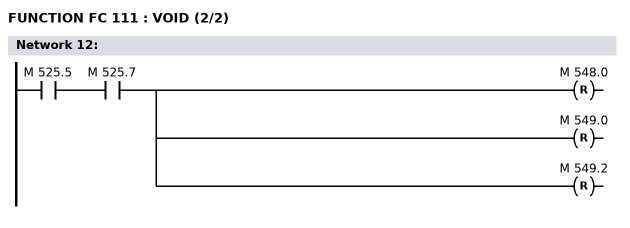

      A     M    525.5;
      A     M    525.7;
      R     M    548.0;
      R     M    549.0;
      R     M    549.2;
END_FUNCTION

FUNCTION_BLOCK FB 112
TITLE =
VERSION : 0.1

BEGIN
NETWORK
TITLE =
